Yaskawa INFORM job: A_ROOF_SIDE_0617_2_PAINT_39.JBI

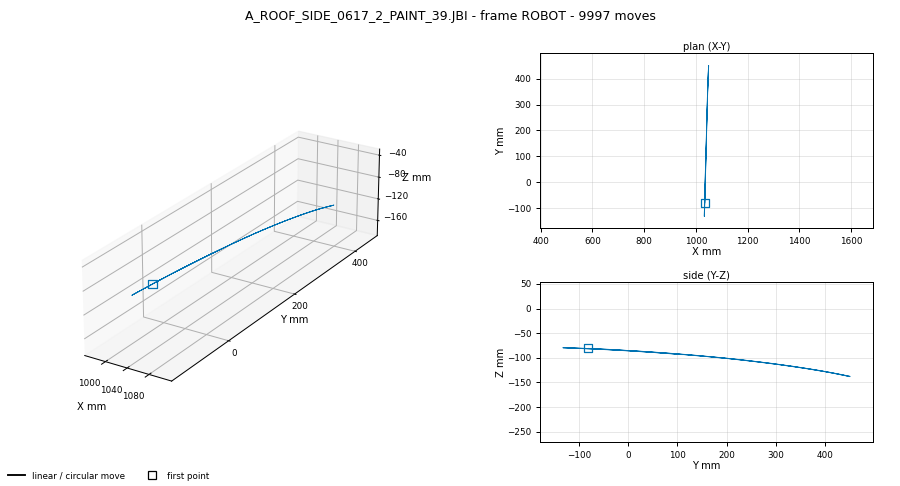
[picture p0: tool path of A_ROOF_SIDE_0617_2_PAINT_39.JBI in frame ROBOT, 9997 of 9997 moves have a stored position in this frame; points joined in program order, loops and branches not executed]
/JOB
//NAME A_ROOF_SIDE_0617_2_PAINT39
//POS
///NPOS 9997,0,0,0,0,0
///TOOL 1
///USER 0
///POSTYPE ROBOT
///RECTAN
///RCONF 1,0,0,0,0,0,0,0,0,0,0,0,0,0,0,0,0,0,0,0,0,0,0,0
C00000=1034.807,-80.393,-80.671,168.125,39.376,157.359
C00001=1034.814,-80.144,-80.681,168.128,39.375,157.359
C00002=1034.820,-79.894,-80.692,168.131,39.374,157.359
C00003=1034.826,-79.644,-80.703,168.134,39.373,157.359
C00004=1034.832,-79.394,-80.715,168.136,39.372,157.359
C00005=1034.838,-79.144,-80.725,168.139,39.372,157.359
C00006=1034.844,-78.895,-80.736,168.142,39.371,157.359
C00007=1034.851,-78.645,-80.747,168.144,39.371,157.359
C00008=1034.856,-78.396,-80.758,168.147,39.370,157.358
C00009=1034.863,-78.145,-80.769,168.150,39.369,157.358
C00010=1034.868,-77.896,-80.780,168.152,39.368,157.358
C00011=1034.875,-77.646,-80.791,168.155,39.368,157.358
C00012=1034.881,-77.397,-80.803,168.157,39.367,157.358
C00013=1034.886,-77.147,-80.814,168.160,39.366,157.358
C00014=1034.893,-76.897,-80.825,168.162,39.365,157.358
C00015=1034.899,-76.648,-80.836,168.165,39.364,157.358
C00016=1034.906,-76.398,-80.846,168.168,39.364,157.358
C00017=1034.911,-76.148,-80.857,168.170,39.363,157.358
C00018=1034.918,-75.899,-80.869,168.173,39.362,157.358
C00019=1034.924,-75.649,-80.880,168.176,39.361,157.358
C00020=1034.930,-75.399,-80.891,168.179,39.361,157.358
C00021=1034.936,-75.150,-80.902,168.181,39.360,157.358
C00022=1034.942,-74.899,-80.914,168.184,39.360,157.358
C00023=1034.948,-74.650,-80.925,168.187,39.359,157.358
C00024=1034.955,-74.400,-80.936,168.189,39.358,157.358
C00025=1034.960,-74.151,-80.947,168.192,39.358,157.358
C00026=1034.967,-73.901,-80.959,168.195,39.357,157.358
C00027=1034.973,-73.652,-80.970,168.196,39.356,157.358
C00028=1034.979,-73.402,-80.981,168.199,39.356,157.358
C00029=1034.985,-73.153,-80.993,168.202,39.355,157.358
C00030=1034.991,-72.902,-81.005,168.204,39.355,157.358
C00031=1034.996,-72.653,-81.016,168.207,39.354,157.358
C00032=1035.002,-72.404,-81.027,168.210,39.354,157.358
C00033=1035.009,-72.154,-81.038,168.212,39.353,157.358
C00034=1035.015,-71.904,-81.049,168.215,39.352,157.358
C00035=1035.020,-71.654,-81.062,168.217,39.352,157.358
C00036=1035.027,-71.404,-81.073,168.220,39.351,157.358
C00037=1035.033,-71.155,-81.085,168.223,39.351,157.358
C00038=1035.039,-70.905,-81.096,168.225,39.350,157.358
C00039=1035.045,-70.656,-81.107,168.228,39.350,157.358
C00040=1035.051,-70.406,-81.119,168.231,39.349,157.358
C00041=1035.057,-70.156,-81.130,168.233,39.348,157.357
C00042=1035.063,-69.907,-81.142,168.236,39.348,157.357
C00043=1035.069,-69.657,-81.153,168.239,39.347,157.357
C00044=1035.076,-69.408,-81.165,168.241,39.347,157.357
C00045=1035.081,-69.158,-81.177,168.244,39.346,157.357
C00046=1035.087,-68.908,-81.188,168.246,39.346,157.357
C00047=1035.094,-68.658,-81.200,168.249,39.345,157.357
C00048=1035.100,-68.375,-81.213,168.251,39.344,157.357
C00049=1035.107,-68.093,-81.226,168.254,39.344,157.357
C00050=1035.114,-67.811,-81.239,168.257,39.343,157.357
C00051=1035.121,-67.528,-81.252,168.260,39.342,157.357
C00052=1035.127,-67.278,-81.264,168.263,39.342,157.357
C00053=1035.133,-67.028,-81.276,168.265,39.341,157.357
C00054=1035.139,-66.778,-81.287,168.268,39.341,157.357
C00055=1035.145,-66.529,-81.299,168.271,39.340,157.357
C00056=1035.152,-66.279,-81.310,168.273,39.340,157.357
C00057=1035.157,-66.029,-81.323,168.276,39.339,157.357
C00058=1035.164,-65.780,-81.334,168.278,39.339,157.357
C00059=1035.170,-65.530,-81.345,168.281,39.338,157.357
C00060=1035.176,-65.281,-81.357,168.284,39.337,157.357
C00061=1035.182,-65.030,-81.369,168.286,39.337,157.357
C00062=1035.188,-64.781,-81.381,168.289,39.336,157.357
C00063=1035.194,-64.532,-81.393,168.292,39.336,157.357
C00064=1035.201,-64.282,-81.404,168.294,39.335,157.357
C00065=1035.206,-64.032,-81.416,168.297,39.335,157.357
C00066=1035.213,-63.783,-81.428,168.299,39.334,157.357
C00067=1035.219,-63.533,-81.439,168.302,39.334,157.357
C00068=1035.226,-63.283,-81.451,168.305,39.333,157.357
C00069=1035.231,-63.034,-81.463,168.307,39.333,157.357
C00070=1035.237,-62.784,-81.475,168.310,39.332,157.357
C00071=1035.244,-62.534,-81.487,168.311,39.331,157.357
C00072=1035.250,-62.285,-81.498,168.314,39.331,157.357
C00073=1035.256,-62.035,-81.511,168.317,39.330,157.357
C00074=1035.262,-61.785,-81.522,168.319,39.330,157.357
C00075=1035.269,-61.536,-81.534,168.322,39.329,157.357
C00076=1035.274,-61.286,-81.546,168.324,39.329,157.357
C00077=1035.281,-61.037,-81.558,168.327,39.328,157.357
C00078=1035.287,-60.787,-81.569,168.330,39.327,157.357
C00079=1035.294,-60.537,-81.581,168.332,39.327,157.357
C00080=1035.299,-60.288,-81.594,168.335,39.326,157.357
C00081=1035.306,-60.038,-81.606,168.338,39.326,157.357
C00082=1035.312,-59.788,-81.617,168.340,39.325,157.357
C00083=1035.318,-59.538,-81.629,168.343,39.325,157.357
C00084=1035.325,-59.289,-81.641,168.345,39.324,157.357
C00085=1035.331,-59.040,-81.653,168.348,39.324,157.357
C00086=1035.337,-58.790,-81.665,168.351,39.323,157.357
C00087=1035.343,-58.540,-81.677,168.353,39.322,157.357
C00088=1035.350,-58.290,-81.689,168.356,39.322,157.357
C00089=1035.356,-58.041,-81.701,168.358,39.321,157.357
C00090=1035.362,-57.791,-81.713,168.361,39.321,157.357
C00091=1035.368,-57.542,-81.725,168.364,39.320,157.357
C00092=1035.375,-57.292,-81.737,168.366,39.320,157.357
C00093=1035.381,-57.042,-81.749,168.369,39.319,157.357
C00094=1035.388,-56.793,-81.761,168.371,39.319,157.357
C00095=1035.394,-56.543,-81.773,168.374,39.318,157.357
C00096=1035.401,-56.294,-81.785,168.375,39.318,157.357
C00097=1035.406,-56.044,-81.797,168.378,39.317,157.357
C00098=1035.412,-55.794,-81.809,168.381,39.316,157.357
C00099=1035.419,-55.545,-81.821,168.383,39.316,157.357
C00100=1035.425,-55.295,-81.833,168.386,39.315,157.357
C00101=1035.432,-55.045,-81.845,168.388,39.315,157.357
C00102=1035.438,-54.796,-81.857,168.391,39.314,157.357
C00103=1035.444,-54.546,-81.870,168.394,39.313,157.357
C00104=1035.451,-54.296,-81.882,168.396,39.313,157.357
C00105=1035.458,-54.047,-81.893,168.399,39.312,157.357
C00106=1035.463,-53.797,-81.906,168.401,39.312,157.357
C00107=1035.469,-53.548,-81.918,168.404,39.311,157.356
C00108=1035.476,-53.298,-81.930,168.407,39.311,157.357
C00109=1035.482,-53.048,-81.942,168.409,39.310,157.356
C00110=1035.489,-52.799,-81.954,168.412,39.310,157.357
C00111=1035.495,-52.549,-81.966,168.414,39.309,157.356
C00112=1035.503,-52.268,-81.980,168.417,39.309,157.356
C00113=1035.510,-51.986,-81.994,168.420,39.308,157.356
C00114=1035.516,-51.705,-82.008,168.423,39.307,157.356
C00115=1035.524,-51.423,-82.021,168.426,39.307,157.356
C00116=1035.530,-51.174,-82.034,168.428,39.306,157.356
C00117=1035.537,-50.924,-82.046,168.431,39.306,157.356
C00118=1035.543,-50.674,-82.058,168.434,39.305,157.356
C00119=1035.549,-50.424,-82.070,168.436,39.305,157.356
C00120=1035.556,-50.175,-82.084,168.439,39.305,157.356
C00121=1035.562,-49.926,-82.096,168.440,39.304,157.356
C00122=1035.568,-49.676,-82.108,168.444,39.304,157.356
C00123=1035.574,-49.426,-82.121,168.446,39.304,157.356
C00124=1035.581,-49.176,-82.133,168.449,39.304,157.357
C00125=1035.587,-48.927,-82.146,168.450,39.303,157.356
C00126=1035.593,-48.677,-82.159,168.453,39.303,157.356
C00127=1035.598,-48.428,-82.171,168.456,39.302,157.357
C00128=1035.605,-48.178,-82.183,168.459,39.302,157.357
C00129=1035.611,-47.929,-82.196,168.460,39.301,157.356
C00130=1035.617,-47.679,-82.208,168.463,39.301,157.357
C00131=1035.624,-47.430,-82.220,168.465,39.301,157.357
C00132=1035.630,-47.180,-82.234,168.468,39.300,157.357
C00133=1035.636,-46.931,-82.246,168.470,39.300,157.357
C00134=1035.642,-46.681,-82.259,168.473,39.300,157.357
C00135=1035.649,-46.432,-82.271,168.475,39.300,157.357
C00136=1035.654,-46.182,-82.284,168.478,39.299,157.357
C00137=1035.660,-45.932,-82.297,168.480,39.299,157.357
C00138=1035.667,-45.683,-82.310,168.483,39.298,157.357
C00139=1035.673,-45.433,-82.322,168.485,39.298,157.357
C00140=1035.679,-45.183,-82.334,168.488,39.297,157.357
C00141=1035.686,-44.933,-82.348,168.490,39.297,157.357
C00142=1035.693,-44.684,-82.360,168.493,39.297,157.357
C00143=1035.698,-44.434,-82.373,168.495,39.297,157.357
C00144=1035.705,-44.185,-82.386,168.498,39.296,157.357
C00145=1035.711,-43.935,-82.398,168.500,39.296,157.357
C00146=1035.718,-43.686,-82.411,168.503,39.296,157.357
C00147=1035.723,-43.436,-82.424,168.505,39.295,157.357
C00148=1035.729,-43.186,-82.436,168.507,39.295,157.357
C00149=1035.736,-42.937,-82.449,168.510,39.294,157.357
C00150=1035.742,-42.687,-82.461,168.512,39.294,157.357
C00151=1035.748,-42.438,-82.475,168.515,39.293,157.357
C00152=1035.754,-42.188,-82.487,168.517,39.293,157.357
C00153=1035.761,-41.939,-82.500,168.520,39.293,157.357
C00154=1035.768,-41.688,-82.513,168.522,39.293,157.357
C00155=1035.774,-41.439,-82.526,168.525,39.292,157.357
C00156=1035.780,-41.189,-82.539,168.527,39.292,157.357
C00157=1035.786,-40.940,-82.552,168.530,39.292,157.357
C00158=1035.793,-40.690,-82.564,168.532,39.292,157.357
C00159=1035.799,-40.441,-82.577,168.535,39.291,157.357
C00160=1035.805,-40.191,-82.590,168.537,39.291,157.357
C00161=1035.812,-39.941,-82.603,168.540,39.290,157.357
C00162=1035.818,-39.691,-82.616,168.542,39.290,157.357
C00163=1035.825,-39.442,-82.629,168.545,39.289,157.357
C00164=1035.831,-39.193,-82.641,168.547,39.289,157.357
C00165=1035.837,-38.943,-82.654,168.550,39.289,157.357
C00166=1035.843,-38.694,-82.668,168.552,39.289,157.357
C00167=1035.849,-38.443,-82.681,168.554,39.288,157.357
C00168=1035.856,-38.194,-82.694,168.557,39.288,157.357
C00169=1035.862,-37.944,-82.706,168.559,39.288,157.357
C00170=1035.868,-37.695,-82.720,168.562,39.287,157.357
C00171=1035.874,-37.446,-82.733,168.564,39.287,157.357
C00172=1035.880,-37.196,-82.745,168.567,39.287,157.357
C00173=1035.886,-36.947,-82.759,168.569,39.287,157.357
C00174=1035.893,-36.697,-82.772,168.571,39.287,157.357
C00175=1035.899,-36.447,-82.786,168.574,39.287,157.357
C00176=1035.906,-36.167,-82.800,168.576,39.286,157.357
C00177=1035.913,-35.885,-82.815,168.579,39.286,157.357
C00178=1035.920,-35.604,-82.830,168.582,39.285,157.357
C00179=1035.928,-35.323,-82.844,168.585,39.285,157.358
C00180=1035.934,-35.074,-82.858,168.587,39.285,157.358
C00181=1035.940,-34.824,-82.871,168.589,39.285,157.358
C00182=1035.946,-34.574,-82.883,168.592,39.285,157.358
C00183=1035.952,-34.325,-82.897,168.594,39.284,157.358
C00184=1035.959,-34.075,-82.910,168.597,39.284,157.358
C00185=1035.964,-33.826,-82.924,168.599,39.284,157.358
C00186=1035.971,-33.576,-82.937,168.601,39.283,157.358
C00187=1035.977,-33.326,-82.950,168.604,39.283,157.358
C00188=1035.983,-33.076,-82.964,168.606,39.283,157.358
C00189=1035.990,-32.827,-82.977,168.609,39.283,157.358
C00190=1035.996,-32.578,-82.990,168.611,39.283,157.358
C00191=1036.002,-32.329,-83.003,168.614,39.282,157.358
C00192=1036.008,-32.078,-83.016,168.616,39.282,157.358
C00193=1036.015,-31.829,-83.030,168.618,39.282,157.358
C00194=1036.021,-31.580,-83.043,168.621,39.282,157.358
C00195=1036.028,-31.330,-83.057,168.623,39.281,157.358
C00196=1036.034,-31.080,-83.070,168.626,39.281,157.358
C00197=1036.040,-30.831,-83.083,168.628,39.281,157.358
C00198=1036.046,-30.582,-83.096,168.630,39.281,157.358
C00199=1036.053,-30.332,-83.110,168.633,39.280,157.358
C00200=1036.059,-30.082,-83.123,168.635,39.280,157.358
C00201=1036.065,-29.833,-83.136,168.637,39.280,157.358
C00202=1036.072,-29.583,-83.149,168.640,39.280,157.358
C00203=1036.078,-29.333,-83.163,168.643,39.280,157.358
C00204=1036.084,-29.084,-83.177,168.645,39.279,157.358
C00205=1036.091,-28.834,-83.190,168.647,39.279,157.358
C00206=1036.097,-28.585,-83.203,168.649,39.279,157.358
C00207=1036.103,-28.335,-83.217,168.652,39.278,157.358
C00208=1036.110,-28.085,-83.230,168.654,39.278,157.358
C00209=1036.116,-27.836,-83.244,168.658,39.278,157.359
C00210=1036.123,-27.586,-83.257,168.660,39.278,157.359
C00211=1036.129,-27.337,-83.271,168.662,39.278,157.359
C00212=1036.135,-27.088,-83.284,168.665,39.277,157.359
C00213=1036.142,-26.838,-83.297,168.667,39.277,157.359
C00214=1036.148,-26.588,-83.311,168.669,39.277,157.359
C00215=1036.154,-26.339,-83.325,168.672,39.277,157.359
C00216=1036.161,-26.089,-83.338,168.674,39.277,157.359
C00217=1036.166,-25.839,-83.352,168.676,39.277,157.359
C00218=1036.172,-25.590,-83.365,168.679,39.276,157.359
C00219=1036.179,-25.341,-83.380,168.681,39.276,157.359
C00220=1036.185,-25.091,-83.394,168.683,39.276,157.359
C00221=1036.192,-24.841,-83.407,168.686,39.276,157.359
C00222=1036.198,-24.592,-83.420,168.688,39.276,157.359
C00223=1036.203,-24.342,-83.434,168.690,39.276,157.359
C00224=1036.210,-24.092,-83.448,168.693,39.275,157.359
C00225=1036.216,-23.843,-83.461,168.695,39.275,157.359
C00226=1036.223,-23.593,-83.476,168.697,39.275,157.359
C00227=1036.229,-23.344,-83.489,168.700,39.275,157.359
C00228=1036.235,-23.095,-83.503,168.702,39.275,157.359
C00229=1036.241,-22.845,-83.517,168.704,39.275,157.359
C00230=1036.248,-22.595,-83.530,168.707,39.274,157.359
C00231=1036.255,-22.346,-83.545,168.709,39.274,157.359
C00232=1036.264,-21.949,-83.566,168.713,39.275,157.360
C00233=1036.274,-21.552,-83.588,168.716,39.274,157.360
C00234=1036.284,-21.155,-83.611,168.720,39.274,157.360
C00235=1036.294,-20.758,-83.632,168.724,39.274,157.360
C00236=1036.304,-20.374,-83.654,168.727,39.274,157.360
C00237=1036.314,-19.990,-83.675,168.731,39.273,157.360
C00238=1036.323,-19.606,-83.696,168.735,39.273,157.360
C00239=1036.333,-19.222,-83.718,168.738,39.273,157.360
C00240=1036.339,-18.973,-83.732,168.740,39.273,157.360
C00241=1036.346,-18.723,-83.745,168.743,39.272,157.360
C00242=1036.352,-18.474,-83.759,168.745,39.272,157.360
C00243=1036.358,-18.224,-83.773,168.747,39.272,157.360
C00244=1036.365,-17.975,-83.787,168.750,39.272,157.360
C00245=1036.371,-17.725,-83.802,168.753,39.272,157.360
C00246=1036.377,-17.476,-83.815,168.755,39.272,157.360
C00247=1036.384,-17.226,-83.829,168.758,39.271,157.360
C00248=1036.390,-16.977,-83.843,168.760,39.271,157.361
C00249=1036.397,-16.727,-83.857,168.762,39.271,157.361
C00250=1036.403,-16.477,-83.872,168.765,39.271,157.361
C00251=1036.409,-16.228,-83.885,168.767,39.271,157.361
C00252=1036.416,-15.979,-83.899,168.769,39.271,157.361
C00253=1036.422,-15.729,-83.913,168.771,39.271,157.361
C00254=1036.429,-15.479,-83.927,168.774,39.270,157.361
C00255=1036.434,-15.230,-83.941,168.776,39.270,157.361
C00256=1036.441,-14.980,-83.955,168.778,39.271,157.361
C00257=1036.447,-14.731,-83.970,168.781,39.270,157.361
C00258=1036.454,-14.481,-83.983,168.783,39.270,157.361
C00259=1036.460,-14.231,-83.998,168.785,39.270,157.361
C00260=1036.466,-13.982,-84.012,168.787,39.270,157.361
C00261=1036.473,-13.733,-84.026,168.790,39.270,157.361
C00262=1036.478,-13.483,-84.040,168.792,39.270,157.361
C00263=1036.485,-13.233,-84.055,168.794,39.270,157.361
C00264=1036.491,-12.985,-84.069,168.796,39.270,157.361
C00265=1036.497,-12.734,-84.083,168.799,39.270,157.361
C00266=1036.504,-12.485,-84.098,168.801,39.270,157.362
C00267=1036.510,-12.235,-84.112,168.803,39.270,157.362
C00268=1036.516,-11.986,-84.127,168.805,39.270,157.362
C00269=1036.522,-11.737,-84.140,168.808,39.270,157.362
C00270=1036.529,-11.487,-84.155,168.810,39.270,157.362
C00271=1036.535,-11.237,-84.170,168.812,39.270,157.362
C00272=1036.541,-10.988,-84.183,168.814,39.269,157.362
C00273=1036.548,-10.738,-84.198,168.818,39.270,157.362
C00274=1036.554,-10.489,-84.213,168.820,39.270,157.362
C00275=1036.560,-10.239,-84.226,168.822,39.270,157.362
C00276=1036.567,-9.990,-84.241,168.824,39.269,157.362
C00277=1036.573,-9.741,-84.256,168.827,39.269,157.362
C00278=1036.579,-9.491,-84.269,168.829,39.269,157.362
C00279=1036.586,-9.241,-84.284,168.831,39.270,157.362
C00280=1036.592,-8.992,-84.299,168.833,39.269,157.362
C00281=1036.598,-8.742,-84.312,168.836,39.269,157.362
C00282=1036.605,-8.493,-84.327,168.838,39.269,157.363
C00283=1036.611,-8.244,-84.342,168.840,39.269,157.363
C00284=1036.617,-7.994,-84.356,168.842,39.269,157.363
C00285=1036.624,-7.744,-84.371,168.844,39.269,157.363
C00286=1036.630,-7.495,-84.385,168.847,39.269,157.363
C00287=1036.637,-7.246,-84.400,168.849,39.269,157.363
C00288=1036.643,-6.995,-84.414,168.851,39.269,157.363
C00289=1036.648,-6.746,-84.428,168.853,39.269,157.363
C00290=1036.656,-6.497,-84.443,168.856,39.268,157.363
C00291=1036.662,-6.247,-84.458,168.858,39.268,157.363
C00292=1036.668,-5.997,-84.472,168.860,39.269,157.363
C00293=1036.675,-5.749,-84.486,168.862,39.269,157.363
C00294=1036.681,-5.499,-84.501,168.865,39.268,157.363
C00295=1036.687,-5.249,-84.516,168.867,39.268,157.363
C00296=1036.694,-5.001,-84.530,168.869,39.268,157.363
C00297=1036.700,-4.750,-84.544,168.871,39.268,157.363
C00298=1036.706,-4.501,-84.559,168.873,39.268,157.363
C00299=1036.713,-4.251,-84.573,168.877,39.268,157.364
C00300=1036.721,-3.968,-84.590,168.879,39.268,157.364
C00301=1036.728,-3.685,-84.607,168.882,39.268,157.364
C00302=1036.734,-3.401,-84.624,168.884,39.268,157.364
C00303=1036.741,-3.118,-84.640,168.887,39.268,157.364
C00304=1036.748,-2.868,-84.655,168.889,39.268,157.364
C00305=1036.754,-2.618,-84.670,168.891,39.268,157.364
C00306=1036.760,-2.369,-84.685,168.893,39.268,157.364
C00307=1036.766,-2.120,-84.699,168.895,39.268,157.364
C00308=1036.773,-1.870,-84.714,168.898,39.268,157.364
C00309=1036.779,-1.620,-84.729,168.900,39.269,157.364
C00310=1036.785,-1.372,-84.744,168.902,39.268,157.364
C00311=1036.791,-1.122,-84.759,168.904,39.268,157.364
C00312=1036.798,-0.872,-84.774,168.906,39.269,157.365
C00313=1036.804,-0.623,-84.789,168.908,39.269,157.365
C00314=1036.810,-0.373,-84.804,168.911,39.268,157.365
C00315=1036.816,-0.124,-84.818,168.914,39.269,157.365
C00316=1036.823,0.126,-84.833,168.916,39.269,157.365
C00317=1036.829,0.375,-84.848,168.918,39.269,157.365
C00318=1036.835,0.625,-84.863,168.920,39.269,157.365
C00319=1036.841,0.874,-84.878,168.922,39.269,157.365
C00320=1036.847,1.124,-84.893,168.924,39.269,157.365
C00321=1036.854,1.373,-84.908,168.927,39.269,157.365
C00322=1036.860,1.623,-84.922,168.929,39.269,157.365
C00323=1036.867,1.872,-84.938,168.931,39.269,157.365
C00324=1036.873,2.121,-84.953,168.933,39.270,157.366
C00325=1036.879,2.371,-84.968,168.935,39.269,157.366
C00326=1036.885,2.620,-84.983,168.937,39.269,157.366
C00327=1036.892,2.870,-84.998,168.940,39.270,157.366
C00328=1036.898,3.120,-85.013,168.942,39.270,157.366
C00329=1036.904,3.370,-85.028,168.944,39.269,157.366
C00330=1036.910,3.619,-85.043,168.946,39.270,157.366
C00331=1036.916,3.868,-85.058,168.948,39.270,157.366
C00332=1036.923,4.117,-85.073,168.950,39.270,157.366
C00333=1036.929,4.367,-85.088,168.953,39.270,157.366
C00334=1036.935,4.617,-85.103,168.956,39.270,157.366
C00335=1036.942,4.866,-85.118,168.958,39.270,157.366
C00336=1036.948,5.116,-85.133,168.960,39.270,157.366
C00337=1036.954,5.364,-85.148,168.962,39.270,157.367
C00338=1036.961,5.614,-85.163,168.964,39.270,157.367
C00339=1036.967,5.863,-85.178,168.966,39.270,157.367
C00340=1036.973,6.113,-85.193,168.969,39.270,157.367
C00341=1036.980,6.362,-85.209,168.971,39.270,157.367
C00342=1036.987,6.612,-85.224,168.973,39.270,157.367
C00343=1036.993,6.861,-85.239,168.975,39.270,157.367
C00344=1036.999,7.111,-85.254,168.977,39.270,157.367
C00345=1037.006,7.360,-85.269,168.979,39.270,157.367
C00346=1037.012,7.610,-85.284,168.981,39.270,157.367
C00347=1037.018,7.860,-85.300,168.984,39.270,157.367
C00348=1037.024,8.109,-85.314,168.986,39.270,157.367
C00349=1037.031,8.358,-85.330,168.988,39.270,157.367
C00350=1037.037,8.607,-85.345,168.991,39.271,157.368
C00351=1037.043,8.857,-85.360,168.993,39.271,157.368
C00352=1037.050,9.106,-85.376,168.995,39.270,157.368
C00353=1037.056,9.356,-85.391,168.997,39.270,157.368
C00354=1037.063,9.605,-85.405,169.000,39.271,157.368
C00355=1037.069,9.854,-85.421,169.002,39.271,157.368
C00356=1037.076,10.104,-85.436,169.004,39.270,157.368
C00357=1037.082,10.354,-85.451,169.006,39.271,157.368
C00358=1037.089,10.603,-85.467,169.008,39.271,157.368
C00359=1037.095,10.853,-85.482,169.010,39.271,157.368
C00360=1037.101,11.102,-85.497,169.012,39.270,157.368
C00361=1037.108,11.352,-85.513,169.014,39.271,157.368
C00362=1037.114,11.601,-85.528,169.017,39.271,157.368
C00363=1037.120,11.851,-85.543,169.019,39.271,157.368
C00364=1037.128,12.136,-85.560,169.021,39.271,157.369
C00365=1037.135,12.421,-85.578,169.024,39.271,157.369
C00366=1037.143,12.706,-85.596,169.026,39.271,157.369
C00367=1037.150,12.992,-85.613,169.029,39.271,157.369
C00368=1037.157,13.241,-85.628,169.032,39.271,157.369
C00369=1037.163,13.491,-85.643,169.034,39.271,157.369
C00370=1037.170,13.740,-85.659,169.036,39.271,157.369
C00371=1037.176,13.990,-85.675,169.038,39.271,157.369
C00372=1037.182,14.239,-85.690,169.040,39.271,157.369
C00373=1037.189,14.489,-85.705,169.042,39.271,157.369
C00374=1037.195,14.738,-85.721,169.044,39.271,157.369
C00375=1037.201,14.988,-85.736,169.046,39.271,157.369
C00376=1037.208,15.237,-85.752,169.048,39.272,157.370
C00377=1037.214,15.486,-85.768,169.051,39.272,157.370
C00378=1037.220,15.736,-85.783,169.053,39.271,157.370
C00379=1037.227,15.985,-85.799,169.055,39.272,157.370
C00380=1037.232,16.235,-85.814,169.057,39.272,157.370
C00381=1037.239,16.484,-85.830,169.059,39.272,157.370
C00382=1037.245,16.734,-85.846,169.061,39.272,157.370
C00383=1037.251,16.983,-85.861,169.063,39.272,157.370
C00384=1037.258,17.232,-85.877,169.066,39.273,157.370
C00385=1037.264,17.482,-85.893,169.068,39.272,157.370
C00386=1037.271,17.732,-85.909,169.070,39.273,157.370
C00387=1037.278,17.981,-85.924,169.072,39.273,157.371
C00388=1037.283,18.231,-85.940,169.074,39.273,157.371
C00389=1037.290,18.480,-85.955,169.077,39.273,157.371
C00390=1037.297,18.729,-85.971,169.079,39.273,157.371
C00391=1037.302,18.979,-85.987,169.081,39.273,157.371
C00392=1037.309,19.228,-86.002,169.083,39.273,157.371
C00393=1037.315,19.477,-86.019,169.085,39.273,157.371
C00394=1037.321,19.727,-86.033,169.087,39.274,157.371
C00395=1037.328,19.976,-86.049,169.089,39.273,157.371
C00396=1037.335,20.226,-86.066,169.091,39.274,157.371
C00397=1037.341,20.475,-86.081,169.093,39.274,157.371
C00398=1037.347,20.725,-86.097,169.095,39.274,157.371
C00399=1037.354,20.974,-86.113,169.098,39.274,157.372
C00400=1037.360,21.223,-86.129,169.100,39.274,157.372
C00401=1037.366,21.473,-86.144,169.102,39.275,157.372
C00402=1037.372,21.722,-86.160,169.104,39.274,157.372
C00403=1037.378,21.971,-86.176,169.106,39.275,157.372
C00404=1037.385,22.221,-86.192,169.109,39.275,157.372
C00405=1037.391,22.471,-86.209,169.111,39.275,157.372
C00406=1037.398,22.720,-86.224,169.113,39.275,157.372
C00407=1037.403,22.970,-86.240,169.115,39.276,157.372
C00408=1037.410,23.219,-86.255,169.117,39.275,157.372
C00409=1037.416,23.468,-86.272,169.119,39.275,157.372
C00410=1037.423,23.717,-86.287,169.121,39.276,157.373
C00411=1037.429,23.966,-86.304,169.123,39.276,157.373
C00412=1037.436,24.217,-86.319,169.126,39.276,157.373
C00413=1037.442,24.466,-86.335,169.128,39.276,157.373
C00414=1037.448,24.715,-86.351,169.130,39.277,157.373
C00415=1037.454,24.964,-86.367,169.132,39.276,157.373
C00416=1037.461,25.213,-86.383,169.134,39.276,157.373
C00417=1037.467,25.463,-86.399,169.136,39.277,157.373
C00418=1037.474,25.713,-86.415,169.138,39.277,157.373
C00419=1037.480,25.962,-86.431,169.140,39.277,157.373
C00420=1037.486,26.211,-86.448,169.142,39.277,157.373
C00421=1037.493,26.461,-86.463,169.144,39.277,157.374
C00422=1037.499,26.711,-86.479,169.146,39.277,157.374
C00423=1037.506,26.960,-86.495,169.149,39.278,157.374
C00424=1037.512,27.209,-86.511,169.151,39.278,157.374
C00425=1037.518,27.459,-86.527,169.153,39.277,157.374
C00426=1037.524,27.708,-86.543,169.156,39.278,157.374
C00427=1037.531,27.958,-86.560,169.158,39.278,157.374
C00428=1037.538,28.244,-86.578,169.160,39.278,157.374
C00429=1037.545,28.531,-86.596,169.162,39.278,157.374
C00430=1037.553,28.817,-86.615,169.165,39.279,157.374
C00431=1037.559,29.104,-86.634,169.167,39.279,157.375
C00432=1037.567,29.353,-86.650,169.169,39.279,157.375
C00433=1037.573,29.603,-86.666,169.171,39.279,157.375
C00434=1037.579,29.852,-86.683,169.173,39.279,157.375
C00435=1037.585,30.101,-86.699,169.175,39.280,157.375
C00436=1037.592,30.351,-86.715,169.177,39.280,157.375
C00437=1037.598,30.601,-86.731,169.179,39.280,157.375
C00438=1037.604,30.850,-86.747,169.182,39.280,157.375
C00439=1037.610,31.099,-86.764,169.184,39.280,157.375
C00440=1037.616,31.348,-86.781,169.186,39.280,157.375
C00441=1037.623,31.598,-86.797,169.188,39.281,157.376
C00442=1037.629,31.847,-86.813,169.190,39.281,157.376
C00443=1037.635,32.096,-86.829,169.192,39.281,157.376
C00444=1037.642,32.346,-86.846,169.194,39.281,157.376
C00445=1037.648,32.596,-86.861,169.196,39.282,157.376
C00446=1037.654,32.845,-86.878,169.198,39.281,157.376
C00447=1037.661,33.094,-86.895,169.200,39.282,157.376
C00448=1037.667,33.344,-86.911,169.202,39.282,157.376
C00449=1037.673,33.593,-86.928,169.204,39.282,157.376
C00450=1037.680,33.842,-86.943,169.207,39.283,157.377
C00451=1037.686,34.092,-86.960,169.209,39.283,157.377
C00452=1037.693,34.341,-86.977,169.211,39.283,157.377
C00453=1037.699,34.590,-86.993,169.213,39.283,157.377
C00454=1037.706,34.840,-87.009,169.215,39.283,157.377
C00455=1037.712,35.089,-87.025,169.217,39.283,157.377
C00456=1037.718,35.339,-87.042,169.219,39.283,157.377
C00457=1037.725,35.588,-87.059,169.221,39.284,157.377
C00458=1037.731,35.837,-87.075,169.223,39.284,157.377
C00459=1037.737,36.086,-87.091,169.225,39.284,157.377
C00460=1037.744,36.336,-87.108,169.227,39.284,157.377
C00461=1037.750,36.585,-87.124,169.229,39.284,157.378
C00462=1037.756,36.835,-87.141,169.231,39.284,157.378
C00463=1037.763,37.085,-87.157,169.234,39.285,157.378
C00464=1037.769,37.333,-87.174,169.236,39.285,157.378
C00465=1037.775,37.583,-87.191,169.238,39.285,157.378
C00466=1037.781,37.833,-87.207,169.240,39.286,157.378
C00467=1037.788,38.081,-87.224,169.242,39.285,157.378
C00468=1037.794,38.332,-87.241,169.244,39.286,157.378
C00469=1037.800,38.581,-87.257,169.246,39.286,157.378
C00470=1037.806,38.830,-87.274,169.248,39.286,157.379
C00471=1037.813,39.080,-87.291,169.250,39.287,157.379
C00472=1037.819,39.329,-87.307,169.252,39.287,157.379
C00473=1037.825,39.578,-87.324,169.254,39.287,157.379
C00474=1037.832,39.828,-87.341,169.257,39.287,157.379
C00475=1037.838,40.076,-87.357,169.259,39.288,157.379
C00476=1037.844,40.326,-87.374,169.261,39.287,157.379
C00477=1037.851,40.575,-87.391,169.263,39.288,157.379
C00478=1037.857,40.825,-87.407,169.265,39.288,157.379
C00479=1037.863,41.075,-87.424,169.267,39.288,157.379
C00480=1037.870,41.323,-87.441,169.269,39.289,157.380
C00481=1037.875,41.573,-87.457,169.271,39.289,157.380
C00482=1037.882,41.822,-87.475,169.273,39.289,157.380
C00483=1037.888,42.072,-87.491,169.275,39.290,157.380
C00484=1037.895,42.321,-87.508,169.277,39.289,157.380
C00485=1037.901,42.570,-87.524,169.280,39.290,157.380
C00486=1037.907,42.819,-87.541,169.282,39.290,157.380
C00487=1037.914,43.069,-87.558,169.284,39.290,157.380
C00488=1037.920,43.318,-87.575,169.286,39.290,157.380
C00489=1037.926,43.568,-87.592,169.288,39.291,157.381
C00490=1037.932,43.817,-87.609,169.290,39.291,157.381
C00491=1037.939,44.067,-87.626,169.292,39.292,157.381
C00492=1037.946,44.353,-87.646,169.294,39.291,157.381
C00493=1037.952,44.639,-87.665,169.296,39.292,157.381
C00494=1037.960,44.926,-87.685,169.298,39.292,157.381
C00495=1037.967,45.213,-87.704,169.302,39.293,157.381
C00496=1037.973,45.461,-87.721,169.304,39.293,157.382
C00497=1037.979,45.711,-87.738,169.305,39.293,157.382
C00498=1037.985,45.960,-87.756,169.307,39.294,157.382
C00499=1037.992,46.210,-87.773,169.309,39.294,157.382
C00500=1037.998,46.459,-87.789,169.311,39.294,157.382
C00501=1038.005,46.709,-87.807,169.313,39.295,157.382
C00502=1038.010,46.958,-87.824,169.315,39.295,157.382
C00503=1038.016,47.207,-87.840,169.317,39.295,157.382
C00504=1038.023,47.456,-87.858,169.320,39.296,157.382
C00505=1038.028,47.706,-87.875,169.322,39.296,157.383
C00506=1038.035,47.956,-87.892,169.324,39.296,157.383
C00507=1038.041,48.204,-87.909,169.326,39.296,157.383
C00508=1038.047,48.454,-87.927,169.328,39.297,157.383
C00509=1038.054,48.703,-87.944,169.330,39.297,157.383
C00510=1038.060,48.953,-87.960,169.332,39.297,157.383
C00511=1038.066,49.202,-87.978,169.334,39.298,157.383
C00512=1038.073,49.451,-87.995,169.336,39.298,157.384
C00513=1038.079,49.701,-88.012,169.337,39.298,157.384
C00514=1038.085,49.950,-88.030,169.340,39.299,157.384
C00515=1038.091,50.199,-88.047,169.342,39.299,157.384
C00516=1038.098,50.449,-88.064,169.344,39.299,157.384
C00517=1038.104,50.697,-88.081,169.346,39.300,157.384
C00518=1038.110,50.948,-88.098,169.348,39.300,157.384
C00519=1038.116,51.196,-88.115,169.350,39.300,157.384
C00520=1038.123,51.446,-88.132,169.352,39.300,157.384
C00521=1038.128,51.695,-88.150,169.354,39.300,157.384
C00522=1038.135,51.944,-88.167,169.356,39.301,157.385
C00523=1038.142,52.194,-88.184,169.358,39.301,157.385
C00524=1038.147,52.443,-88.201,169.360,39.301,157.385
C00525=1038.154,52.693,-88.219,169.363,39.302,157.385
C00526=1038.161,52.942,-88.236,169.365,39.302,157.385
C00527=1038.167,53.191,-88.254,169.367,39.302,157.385
C00528=1038.173,53.440,-88.271,169.369,39.302,157.385
C00529=1038.179,53.690,-88.289,169.371,39.303,157.385
C00530=1038.185,53.939,-88.305,169.373,39.303,157.386
C00531=1038.192,54.189,-88.322,169.375,39.303,157.386
C00532=1038.198,54.438,-88.340,169.376,39.304,157.386
C00533=1038.204,54.687,-88.357,169.378,39.304,157.386
C00534=1038.211,54.936,-88.374,169.381,39.304,157.386
C00535=1038.217,55.185,-88.392,169.383,39.304,157.386
C00536=1038.223,55.435,-88.409,169.385,39.305,157.386
C00537=1038.230,55.684,-88.427,169.387,39.305,157.386
C00538=1038.236,55.933,-88.444,169.389,39.305,157.386
C00539=1038.243,56.183,-88.462,169.391,39.305,157.387
C00540=1038.250,56.432,-88.479,169.393,39.305,157.387
C00541=1038.255,56.681,-88.496,169.395,39.306,157.387
C00542=1038.262,56.931,-88.514,169.397,39.306,157.387
C00543=1038.267,57.180,-88.531,169.399,39.306,157.387
C00544=1038.274,57.429,-88.549,169.401,39.307,157.387
C00545=1038.281,57.679,-88.565,169.404,39.307,157.387
C00546=1038.286,57.928,-88.583,169.406,39.307,157.387
C00547=1038.293,58.178,-88.600,169.408,39.307,157.387
C00548=1038.300,58.427,-88.618,169.410,39.307,157.388
C00549=1038.306,58.676,-88.636,169.412,39.308,157.388
C00550=1038.313,58.925,-88.653,169.414,39.308,157.388
C00551=1038.320,59.174,-88.671,169.416,39.308,157.388
C00552=1038.325,59.423,-88.688,169.418,39.309,157.388
C00553=1038.332,59.673,-88.705,169.419,39.309,157.388
C00554=1038.338,59.923,-88.723,169.421,39.309,157.388
C00555=1038.345,60.172,-88.741,169.423,39.309,157.388
C00556=1038.352,60.458,-88.761,169.427,39.309,157.388
C00557=1038.360,60.745,-88.781,169.429,39.310,157.389
C00558=1038.366,61.031,-88.801,169.431,39.310,157.389
C00559=1038.374,61.317,-88.821,169.433,39.310,157.389
C00560=1038.380,61.566,-88.838,169.435,39.311,157.389
C00561=1038.387,61.815,-88.856,169.437,39.310,157.389
C00562=1038.393,62.065,-88.874,169.439,39.311,157.389
C00563=1038.400,62.315,-88.891,169.441,39.311,157.389
C00564=1038.406,62.564,-88.908,169.443,39.311,157.389
C00565=1038.413,62.812,-88.926,169.445,39.311,157.389
C00566=1038.420,63.062,-88.944,169.447,39.312,157.390
C00567=1038.426,63.312,-88.962,169.450,39.312,157.390
C00568=1038.432,63.560,-88.979,169.452,39.312,157.390
C00569=1038.438,63.810,-88.997,169.454,39.312,157.390
C00570=1038.445,64.059,-89.014,169.456,39.312,157.390
C00571=1038.451,64.309,-89.033,169.458,39.313,157.390
C00572=1038.457,64.558,-89.050,169.460,39.313,157.390
C00573=1038.464,64.807,-89.068,169.462,39.314,157.390
C00574=1038.470,65.057,-89.085,169.464,39.314,157.390
C00575=1038.476,65.306,-89.104,169.466,39.314,157.391
C00576=1038.483,65.555,-89.121,169.468,39.315,157.391
C00577=1038.489,65.804,-89.139,169.470,39.315,157.391
C00578=1038.495,66.053,-89.158,169.472,39.315,157.391
C00579=1038.502,66.303,-89.175,169.474,39.316,157.391
C00580=1038.508,66.552,-89.193,169.476,39.315,157.391
C00581=1038.514,66.802,-89.211,169.478,39.316,157.391
C00582=1038.521,67.050,-89.229,169.480,39.316,157.391
C00583=1038.527,67.300,-89.246,169.482,39.317,157.392
C00584=1038.532,67.549,-89.264,169.484,39.317,157.392
C00585=1038.539,67.798,-89.283,169.486,39.317,157.392
C00586=1038.546,68.048,-89.300,169.489,39.318,157.392
C00587=1038.552,68.297,-89.319,169.491,39.318,157.392
C00588=1038.558,68.546,-89.336,169.493,39.318,157.392
C00589=1038.565,68.795,-89.354,169.494,39.319,157.392
C00590=1038.571,69.045,-89.372,169.496,39.319,157.393
C00591=1038.577,69.294,-89.390,169.498,39.319,157.393
C00592=1038.584,69.543,-89.409,169.500,39.320,157.393
C00593=1038.589,69.792,-89.426,169.502,39.320,157.393
C00594=1038.596,70.042,-89.444,169.504,39.320,157.393
C00595=1038.602,70.291,-89.462,169.506,39.320,157.393
C00596=1038.608,70.541,-89.480,169.509,39.321,157.393
C00597=1038.615,70.790,-89.499,169.511,39.321,157.393
C00598=1038.620,71.039,-89.517,169.513,39.322,157.394
C00599=1038.627,71.288,-89.535,169.515,39.322,157.394
C00600=1038.633,71.538,-89.553,169.517,39.322,157.394
C00601=1038.640,71.787,-89.571,169.518,39.323,157.394
C00602=1038.646,72.036,-89.589,169.520,39.323,157.394
C00603=1038.652,72.285,-89.607,169.522,39.323,157.394
C00604=1038.658,72.534,-89.625,169.524,39.324,157.394
C00605=1038.665,72.784,-89.644,169.527,39.324,157.394
C00606=1038.671,73.033,-89.662,169.529,39.325,157.395
C00607=1038.677,73.282,-89.681,169.531,39.324,157.395
C00608=1038.683,73.532,-89.698,169.533,39.325,157.395
C00609=1038.689,73.781,-89.717,169.535,39.325,157.395
C00610=1038.696,74.030,-89.735,169.537,39.326,157.395
C00611=1038.702,74.279,-89.753,169.539,39.326,157.395
C00612=1038.709,74.528,-89.771,169.540,39.326,157.395
C00613=1038.715,74.778,-89.789,169.543,39.327,157.395
C00614=1038.721,75.027,-89.808,169.545,39.327,157.396
C00615=1038.728,75.276,-89.827,169.547,39.327,157.396
C00616=1038.733,75.525,-89.844,169.549,39.328,157.396
C00617=1038.740,75.774,-89.863,169.551,39.328,157.396
C00618=1038.746,76.024,-89.881,169.553,39.329,157.396
C00619=1038.752,76.273,-89.899,169.555,39.328,157.396
C00620=1038.760,76.559,-89.920,169.557,39.329,157.396
C00621=1038.767,76.845,-89.942,169.559,39.329,157.396
C00622=1038.774,77.132,-89.962,169.563,39.330,157.397
C00623=1038.781,77.418,-89.984,169.565,39.330,157.397
C00624=1038.788,77.667,-90.002,169.567,39.331,157.397
C00625=1038.794,77.915,-90.021,169.569,39.331,157.397
C00626=1038.800,78.165,-90.039,169.570,39.331,157.397
C00627=1038.806,78.414,-90.057,169.572,39.332,157.397
C00628=1038.813,78.663,-90.076,169.574,39.332,157.397
C00629=1038.819,78.913,-90.094,169.576,39.333,157.398
C00630=1038.825,79.162,-90.112,169.578,39.333,157.398
C00631=1038.831,79.412,-90.132,169.581,39.333,157.398
C00632=1038.837,79.661,-90.150,169.583,39.334,157.398
C00633=1038.844,79.910,-90.169,169.585,39.334,157.398
C00634=1038.850,80.160,-90.187,169.587,39.335,157.398
C00635=1038.856,80.408,-90.205,169.589,39.335,157.398
C00636=1038.861,80.658,-90.224,169.590,39.336,157.399
C00637=1038.868,80.907,-90.243,169.592,39.335,157.399
C00638=1038.874,81.156,-90.262,169.594,39.336,157.399
C00639=1038.881,81.405,-90.280,169.597,39.336,157.399
C00640=1038.887,81.655,-90.298,169.599,39.337,157.399
C00641=1038.893,81.904,-90.317,169.601,39.337,157.399
C00642=1038.899,82.153,-90.336,169.603,39.338,157.399
C00643=1038.905,82.402,-90.355,169.605,39.338,157.400
C00644=1038.912,82.651,-90.373,169.607,39.338,157.400
C00645=1038.918,82.901,-90.392,169.609,39.339,157.400
C00646=1038.925,83.150,-90.411,169.610,39.339,157.400
C00647=1038.930,83.399,-90.430,169.613,39.340,157.400
C00648=1038.937,83.648,-90.449,169.615,39.340,157.400
C00649=1038.943,83.898,-90.467,169.617,39.340,157.400
C00650=1038.949,84.147,-90.485,169.619,39.341,157.401
C00651=1038.956,84.396,-90.504,169.621,39.341,157.401
C00652=1038.961,84.646,-90.523,169.623,39.342,157.401
C00653=1038.968,84.895,-90.542,169.625,39.342,157.401
C00654=1038.974,85.144,-90.560,169.627,39.342,157.401
C00655=1038.981,85.393,-90.579,169.630,39.342,157.401
C00656=1038.987,85.642,-90.598,169.632,39.343,157.401
C00657=1038.993,85.892,-90.617,169.634,39.343,157.402
C00658=1038.999,86.141,-90.636,169.635,39.344,157.402
C00659=1039.006,86.390,-90.654,169.637,39.344,157.402
C00660=1039.012,86.639,-90.673,169.639,39.344,157.402
C00661=1039.018,86.888,-90.692,169.641,39.345,157.402
C00662=1039.024,87.138,-90.711,169.643,39.345,157.402
C00663=1039.031,87.387,-90.729,169.646,39.346,157.402
C00664=1039.037,87.636,-90.748,169.648,39.346,157.402
C00665=1039.043,87.885,-90.767,169.650,39.346,157.403
C00666=1039.049,88.134,-90.786,169.652,39.347,157.403
C00667=1039.055,88.383,-90.805,169.654,39.347,157.403
C00668=1039.062,88.633,-90.823,169.656,39.348,157.403
C00669=1039.068,88.882,-90.842,169.658,39.347,157.403
C00670=1039.075,89.131,-90.861,169.660,39.348,157.403
C00671=1039.080,89.380,-90.880,169.661,39.348,157.403
C00672=1039.087,89.630,-90.899,169.664,39.349,157.404
C00673=1039.094,89.879,-90.918,169.666,39.349,157.404
C00674=1039.101,90.128,-90.937,169.668,39.349,157.404
C00675=1039.106,90.377,-90.956,169.670,39.350,157.404
C00676=1039.113,90.626,-90.975,169.672,39.350,157.404
C00677=1039.118,90.876,-90.994,169.674,39.351,157.404
C00678=1039.125,91.125,-91.013,169.676,39.351,157.404
C00679=1039.131,91.374,-91.033,169.678,39.352,157.405
C00680=1039.137,91.623,-91.051,169.681,39.352,157.405
C00681=1039.143,91.872,-91.071,169.683,39.353,157.405
C00682=1039.149,92.121,-91.089,169.684,39.353,157.405
C00683=1039.155,92.371,-91.108,169.686,39.353,157.405
C00684=1039.163,92.656,-91.131,169.689,39.354,157.405
C00685=1039.170,92.943,-91.152,169.691,39.355,157.406
C00686=1039.177,93.228,-91.175,169.693,39.355,157.406
C00687=1039.184,93.515,-91.196,169.696,39.356,157.406
C00688=1039.190,93.764,-91.216,169.698,39.356,157.406
C00689=1039.197,94.013,-91.235,169.700,39.356,157.406
C00690=1039.202,94.262,-91.254,169.702,39.356,157.406
C00691=1039.209,94.511,-91.273,169.704,39.357,157.406
C00692=1039.215,94.760,-91.293,169.706,39.357,157.407
C00693=1039.221,95.009,-91.311,169.708,39.358,157.407
C00694=1039.227,95.259,-91.331,169.711,39.358,157.407
C00695=1039.234,95.508,-91.350,169.712,39.359,157.407
C00696=1039.240,95.757,-91.370,169.714,39.359,157.407
C00697=1039.246,96.007,-91.389,169.716,39.359,157.407
C00698=1039.252,96.255,-91.408,169.718,39.360,157.407
C00699=1039.258,96.505,-91.428,169.720,39.360,157.408
C00700=1039.264,96.754,-91.446,169.722,39.361,157.408
C00701=1039.271,97.003,-91.466,169.724,39.361,157.408
C00702=1039.277,97.252,-91.485,169.727,39.362,157.408
C00703=1039.283,97.502,-91.504,169.729,39.362,157.408
C00704=1039.290,97.750,-91.524,169.731,39.363,157.408
C00705=1039.296,98.000,-91.543,169.733,39.363,157.408
C00706=1039.302,98.249,-91.562,169.735,39.363,157.409
C00707=1039.309,98.498,-91.582,169.737,39.364,157.409
C00708=1039.315,98.748,-91.601,169.739,39.364,157.409
C00709=1039.321,98.996,-91.621,169.740,39.365,157.409
C00710=1039.327,99.245,-91.639,169.743,39.365,157.409
C00711=1039.333,99.494,-91.659,169.745,39.366,157.409
C00712=1039.340,99.744,-91.679,169.747,39.365,157.409
C00713=1039.346,99.994,-91.697,169.749,39.366,157.410
C00714=1039.352,100.242,-91.717,169.751,39.366,157.410
C00715=1039.359,100.491,-91.736,169.753,39.367,157.410
C00716=1039.365,100.740,-91.756,169.755,39.367,157.410
C00717=1039.371,100.990,-91.776,169.757,39.368,157.410
C00718=1039.377,101.239,-91.796,169.760,39.368,157.410
C00719=1039.384,101.488,-91.815,169.762,39.369,157.410
C00720=1039.389,101.737,-91.834,169.764,39.369,157.411
C00721=1039.395,101.986,-91.854,169.766,39.370,157.411
C00722=1039.402,102.236,-91.874,169.768,39.370,157.411
C00723=1039.408,102.485,-91.894,169.769,39.371,157.411
C00724=1039.414,102.734,-91.912,169.771,39.371,157.411
C00725=1039.420,102.983,-91.932,169.774,39.372,157.411
C00726=1039.426,103.232,-91.952,169.776,39.372,157.412
C00727=1039.432,103.482,-91.972,169.778,39.373,157.412
C00728=1039.438,103.731,-91.992,169.780,39.373,157.412
C00729=1039.445,103.979,-92.011,169.782,39.374,157.412
C00730=1039.451,104.229,-92.030,169.784,39.374,157.412
C00731=1039.457,104.478,-92.051,169.786,39.375,157.412
C00732=1039.463,104.728,-92.070,169.789,39.375,157.413
C00733=1039.469,104.976,-92.090,169.791,39.376,157.413
C00734=1039.475,105.225,-92.110,169.793,39.376,157.413
C00735=1039.482,105.475,-92.129,169.795,39.377,157.413
C00736=1039.488,105.724,-92.149,169.796,39.377,157.413
C00737=1039.494,105.973,-92.169,169.798,39.378,157.413
C00738=1039.501,106.222,-92.189,169.800,39.378,157.414
C00739=1039.506,106.472,-92.208,169.802,39.378,157.414
C00740=1039.513,106.720,-92.228,169.805,39.379,157.414
C00741=1039.519,106.969,-92.248,169.807,39.379,157.414
C00742=1039.525,107.219,-92.267,169.809,39.379,157.414
C00743=1039.531,107.468,-92.287,169.811,39.380,157.414
C00744=1039.537,107.717,-92.307,169.813,39.380,157.414
C00745=1039.544,107.966,-92.328,169.815,39.381,157.415
C00746=1039.550,108.215,-92.346,169.817,39.381,157.415
C00747=1039.556,108.464,-92.366,169.820,39.382,157.415
C00748=1039.563,108.750,-92.389,169.822,39.382,157.415
C00749=1039.571,109.036,-92.412,169.824,39.383,157.415
C00750=1039.578,109.322,-92.435,169.827,39.383,157.415
C00751=1039.585,109.608,-92.457,169.829,39.384,157.416
C00752=1039.591,109.857,-92.477,169.831,39.384,157.416
C00753=1039.598,110.107,-92.497,169.834,39.385,157.416
C00754=1039.604,110.355,-92.517,169.836,39.385,157.416
C00755=1039.610,110.604,-92.537,169.838,39.386,157.416
C00756=1039.616,110.854,-92.558,169.840,39.386,157.416
C00757=1039.622,111.103,-92.577,169.842,39.387,157.417
C00758=1039.628,111.352,-92.597,169.844,39.387,157.417
C00759=1039.635,111.601,-92.617,169.846,39.388,157.417
C00760=1039.641,111.850,-92.637,169.848,39.388,157.417
C00761=1039.647,112.100,-92.657,169.850,39.389,157.417
C00762=1039.653,112.349,-92.677,169.852,39.389,157.417
C00763=1039.659,112.597,-92.697,169.854,39.390,157.418
C00764=1039.666,112.847,-92.718,169.856,39.390,157.418
C00765=1039.672,113.096,-92.738,169.858,39.391,157.418
C00766=1039.678,113.345,-92.758,169.860,39.391,157.418
C00767=1039.684,113.594,-92.778,169.863,39.392,157.418
C00768=1039.690,113.843,-92.798,169.865,39.392,157.418
C00769=1039.696,114.092,-92.818,169.867,39.393,157.419
C00770=1039.702,114.341,-92.839,169.869,39.394,157.419
C00771=1039.708,114.590,-92.859,169.871,39.394,157.419
C00772=1039.714,114.839,-92.879,169.873,39.395,157.419
C00773=1039.720,115.089,-92.900,169.876,39.395,157.419
C00774=1039.726,115.338,-92.920,169.878,39.396,157.419
C00775=1039.732,115.587,-92.940,169.880,39.396,157.420
C00776=1039.739,115.836,-92.960,169.882,39.397,157.420
C00777=1039.744,116.085,-92.980,169.883,39.398,157.420
C00778=1039.750,116.335,-93.001,169.885,39.398,157.420
C00779=1039.756,116.584,-93.021,169.888,39.399,157.420
C00780=1039.763,116.832,-93.041,169.890,39.399,157.421
C00781=1039.769,117.082,-93.062,169.892,39.400,157.421
C00782=1039.775,117.330,-93.082,169.894,39.400,157.421
C00783=1039.781,117.580,-93.103,169.896,39.401,157.421
C00784=1039.787,117.829,-93.123,169.898,39.401,157.421
C00785=1039.792,118.078,-93.143,169.901,39.402,157.421
C00786=1039.799,118.327,-93.163,169.903,39.403,157.422
C00787=1039.805,118.576,-93.184,169.905,39.403,157.422
C00788=1039.811,118.825,-93.205,169.907,39.404,157.422
C00789=1039.817,119.074,-93.225,169.909,39.404,157.422
C00790=1039.824,119.324,-93.245,169.911,39.405,157.422
C00791=1039.830,119.572,-93.265,169.913,39.405,157.422
C00792=1039.835,119.821,-93.287,169.916,39.406,157.423
C00793=1039.842,120.071,-93.307,169.918,39.406,157.423
C00794=1039.848,120.319,-93.327,169.920,39.407,157.423
C00795=1039.854,120.569,-93.348,169.922,39.408,157.423
C00796=1039.860,120.817,-93.368,169.924,39.408,157.423
C00797=1039.867,121.067,-93.389,169.926,39.409,157.424
C00798=1039.872,121.316,-93.409,169.929,39.409,157.424
C00799=1039.879,121.565,-93.430,169.931,39.410,157.424
C00800=1039.885,121.814,-93.450,169.933,39.410,157.424
C00801=1039.891,122.063,-93.471,169.935,39.411,157.424
C00802=1039.897,122.312,-93.491,169.937,39.411,157.424
C00803=1039.903,122.562,-93.512,169.938,39.412,157.425
C00804=1039.910,122.810,-93.532,169.941,39.413,157.425
C00805=1039.915,123.060,-93.553,169.943,39.413,157.425
C00806=1039.921,123.309,-93.573,169.945,39.414,157.425
C00807=1039.928,123.558,-93.594,169.947,39.414,157.425
C00808=1039.934,123.807,-93.615,169.949,39.415,157.425
C00809=1039.940,124.056,-93.635,169.951,39.415,157.426
C00810=1039.946,124.304,-93.656,169.953,39.416,157.426
C00811=1039.952,124.554,-93.677,169.956,39.416,157.426
C00812=1039.959,124.840,-93.700,169.959,39.416,157.426
C00813=1039.967,125.126,-93.724,169.961,39.418,157.426
C00814=1039.974,125.412,-93.747,169.963,39.418,157.427
C00815=1039.981,125.697,-93.771,169.966,39.418,157.427
C00816=1039.988,125.946,-93.792,169.968,39.419,157.427
C00817=1039.994,126.196,-93.812,169.971,39.419,157.427
C00818=1039.999,126.445,-93.833,169.973,39.420,157.427
C00819=1040.006,126.694,-93.854,169.975,39.420,157.427
C00820=1040.012,126.942,-93.874,169.977,39.421,157.428
C00821=1040.018,127.192,-93.895,169.979,39.422,157.428
C00822=1040.025,127.441,-93.916,169.981,39.422,157.428
C00823=1040.031,127.689,-93.936,169.984,39.423,157.428
C00824=1040.037,127.939,-93.957,169.986,39.423,157.428
C00825=1040.043,128.187,-93.978,169.988,39.424,157.429
C00826=1040.050,128.437,-93.998,169.990,39.424,157.429
C00827=1040.056,128.687,-94.019,169.992,39.425,157.429
C00828=1040.062,128.935,-94.040,169.994,39.425,157.429
C00829=1040.068,129.185,-94.061,169.997,39.426,157.429
C00830=1040.075,129.434,-94.082,169.999,39.426,157.429
C00831=1040.081,129.682,-94.102,170.001,39.427,157.430
C00832=1040.087,129.932,-94.123,170.003,39.427,157.430
C00833=1040.093,130.180,-94.144,170.005,39.428,157.430
C00834=1040.100,130.429,-94.164,170.007,39.428,157.430
C00835=1040.106,130.678,-94.186,170.009,39.429,157.430
C00836=1040.112,130.927,-94.206,170.012,39.430,157.430
C00837=1040.118,131.177,-94.228,170.014,39.430,157.431
C00838=1040.125,131.426,-94.248,170.016,39.431,157.431
C00839=1040.131,131.675,-94.269,170.018,39.431,157.431
C00840=1040.137,131.924,-94.291,170.020,39.432,157.431
C00841=1040.143,132.173,-94.311,170.023,39.433,157.431
C00842=1040.149,132.422,-94.333,170.025,39.433,157.432
C00843=1040.156,132.671,-94.354,170.027,39.434,157.432
C00844=1040.162,132.920,-94.374,170.029,39.434,157.432
C00845=1040.167,133.169,-94.396,170.031,39.435,157.432
C00846=1040.174,133.418,-94.417,170.034,39.436,157.432
C00847=1040.180,133.667,-94.438,170.037,39.436,157.433
C00848=1040.185,133.916,-94.459,170.039,39.437,157.433
C00849=1040.192,134.165,-94.480,170.041,39.437,157.433
C00850=1040.199,134.414,-94.502,170.043,39.438,157.433
C00851=1040.204,134.663,-94.523,170.045,39.439,157.433
C00852=1040.211,134.912,-94.543,170.047,39.439,157.434
C00853=1040.217,135.162,-94.565,170.050,39.440,157.434
C00854=1040.222,135.410,-94.586,170.052,39.440,157.434
C00855=1040.229,135.659,-94.607,170.054,39.441,157.434
C00856=1040.235,135.909,-94.628,170.056,39.442,157.434
C00857=1040.241,136.157,-94.649,170.058,39.442,157.434
C00858=1040.248,136.406,-94.670,170.060,39.443,157.435
C00859=1040.254,136.655,-94.692,170.063,39.443,157.435
C00860=1040.260,136.905,-94.714,170.065,39.444,157.435
C00861=1040.266,137.153,-94.735,170.067,39.445,157.435
C00862=1040.272,137.403,-94.755,170.069,39.445,157.435
C00863=1040.278,137.652,-94.777,170.071,39.446,157.436
C00864=1040.284,137.900,-94.798,170.074,39.447,157.436
C00865=1040.290,138.149,-94.820,170.076,39.447,157.436
C00866=1040.297,138.398,-94.841,170.078,39.448,157.436
C00867=1040.303,138.648,-94.863,170.081,39.448,157.436
C00868=1040.309,138.896,-94.884,170.083,39.449,157.437
C00869=1040.315,139.145,-94.905,170.085,39.450,157.437
C00870=1040.322,139.394,-94.926,170.088,39.450,157.437
C00871=1040.328,139.644,-94.947,170.090,39.451,157.437
C00872=1040.333,139.893,-94.969,170.092,39.452,157.437
C00873=1040.339,140.142,-94.990,170.094,39.452,157.438
C00874=1040.345,140.391,-95.012,170.096,39.453,157.438
C00875=1040.352,140.640,-95.034,170.099,39.454,157.438
C00876=1040.358,140.925,-95.059,170.101,39.454,157.438
C00877=1040.366,141.211,-95.083,170.104,39.455,157.439
C00878=1040.372,141.496,-95.108,170.106,39.456,157.439
C00879=1040.380,141.782,-95.133,170.108,39.457,157.439
C00880=1040.385,142.031,-95.154,170.112,39.457,157.439
C00881=1040.391,142.280,-95.176,170.114,39.458,157.439
C00882=1040.397,142.529,-95.197,170.116,39.459,157.440
C00883=1040.404,142.778,-95.218,170.118,39.459,157.440
C00884=1040.411,143.027,-95.240,170.120,39.460,157.440
C00885=1040.416,143.276,-95.261,170.123,39.461,157.440
C00886=1040.422,143.525,-95.283,170.125,39.461,157.440
C00887=1040.428,143.774,-95.305,170.127,39.462,157.441
C00888=1040.435,144.023,-95.327,170.129,39.463,157.441
C00889=1040.441,144.272,-95.349,170.131,39.463,157.441
C00890=1040.447,144.520,-95.370,170.133,39.464,157.441
C00891=1040.453,144.770,-95.391,170.136,39.465,157.442
C00892=1040.459,145.019,-95.413,170.139,39.465,157.442
C00893=1040.465,145.268,-95.435,170.141,39.466,157.442
C00894=1040.471,145.517,-95.456,170.143,39.466,157.442
C00895=1040.478,145.766,-95.479,170.145,39.467,157.442
C00896=1040.484,146.015,-95.500,170.148,39.468,157.442
C00897=1040.489,146.264,-95.522,170.150,39.468,157.443
C00898=1040.496,146.513,-95.543,170.152,39.470,157.443
C00899=1040.502,146.762,-95.565,170.154,39.470,157.443
C00900=1040.508,147.011,-95.587,170.156,39.470,157.443
C00901=1040.514,147.260,-95.609,170.159,39.472,157.444
C00902=1040.521,147.509,-95.631,170.162,39.472,157.444
C00903=1040.527,147.758,-95.652,170.164,39.473,157.444
C00904=1040.533,148.007,-95.675,170.166,39.474,157.444
C00905=1040.539,148.255,-95.696,170.168,39.474,157.444
C00906=1040.545,148.504,-95.717,170.171,39.475,157.445
C00907=1040.551,148.753,-95.740,170.173,39.476,157.445
C00908=1040.558,149.002,-95.761,170.175,39.477,157.445
C00909=1040.563,149.252,-95.784,170.177,39.477,157.445
C00910=1040.569,149.500,-95.806,170.179,39.478,157.445
C00911=1040.576,149.750,-95.828,170.183,39.479,157.446
C00912=1040.582,149.999,-95.849,170.185,39.479,157.446
C00913=1040.588,150.247,-95.871,170.187,39.480,157.446
C00914=1040.594,150.496,-95.893,170.189,39.481,157.446
C00915=1040.599,150.745,-95.915,170.192,39.482,157.447
C00916=1040.606,150.994,-95.937,170.194,39.482,157.447
C00917=1040.612,151.243,-95.959,170.196,39.483,157.447
C00918=1040.618,151.492,-95.981,170.198,39.484,157.447
C00919=1040.624,151.741,-96.004,170.201,39.484,157.448
C00920=1040.630,151.990,-96.026,170.204,39.485,157.448
C00921=1040.636,152.239,-96.048,170.206,39.486,157.448
C00922=1040.643,152.488,-96.069,170.208,39.487,157.448
C00923=1040.649,152.737,-96.092,170.210,39.487,157.448
C00924=1040.654,152.986,-96.114,170.212,39.488,157.449
C00925=1040.661,153.235,-96.136,170.215,39.489,157.449
C00926=1040.667,153.484,-96.158,170.218,39.489,157.449
C00927=1040.674,153.733,-96.180,170.220,39.490,157.449
C00928=1040.680,153.982,-96.202,170.222,39.491,157.450
C00929=1040.685,154.231,-96.225,170.224,39.492,157.450
C00930=1040.692,154.480,-96.246,170.227,39.492,157.450
C00931=1040.698,154.729,-96.269,170.229,39.494,157.450
C00932=1040.703,154.977,-96.291,170.231,39.494,157.450
C00933=1040.709,155.226,-96.313,170.234,39.495,157.451
C00934=1040.716,155.475,-96.335,170.236,39.496,157.451
C00935=1040.721,155.724,-96.358,170.239,39.497,157.451
C00936=1040.728,155.973,-96.380,170.241,39.497,157.451
C00937=1040.734,156.221,-96.402,170.243,39.498,157.452
C00938=1040.740,156.471,-96.425,170.245,39.499,157.452
C00939=1040.746,156.719,-96.447,170.249,39.500,157.452
C00940=1040.753,157.005,-96.472,170.251,39.500,157.452
C00941=1040.761,157.290,-96.498,170.253,39.501,157.453
C00942=1040.767,157.576,-96.524,170.256,39.502,157.453
C00943=1040.774,157.861,-96.550,170.259,39.503,157.453
C00944=1040.780,158.110,-96.572,170.262,39.504,157.453
C00945=1040.787,158.359,-96.594,170.264,39.505,157.454
C00946=1040.792,158.608,-96.617,170.266,39.505,157.454
C00947=1040.799,158.856,-96.639,170.268,39.506,157.454
C00948=1040.804,159.106,-96.661,170.271,39.507,157.454
C00949=1040.811,159.354,-96.684,170.274,39.508,157.455
C00950=1040.817,159.603,-96.706,170.276,39.508,157.455
C00951=1040.823,159.852,-96.728,170.278,39.509,157.455
C00952=1040.829,160.101,-96.751,170.280,39.510,157.455
C00953=1040.835,160.351,-96.774,170.283,39.511,157.456
C00954=1040.842,160.599,-96.796,170.285,39.512,157.456
C00955=1040.848,160.848,-96.819,170.288,39.513,157.456
C00956=1040.853,161.097,-96.842,170.290,39.514,157.456
C00957=1040.859,161.346,-96.865,170.293,39.515,157.457
C00958=1040.865,161.595,-96.887,170.295,39.516,157.457
C00959=1040.871,161.844,-96.910,170.297,39.516,157.457
C00960=1040.877,162.093,-96.933,170.299,39.517,157.457
C00961=1040.882,162.342,-96.956,170.303,39.518,157.458
C00962=1040.888,162.591,-96.979,170.305,39.519,157.458
C00963=1040.895,162.839,-97.001,170.307,39.520,157.458
C00964=1040.900,163.088,-97.024,170.309,39.521,157.458
C00965=1040.906,163.337,-97.047,170.312,39.522,157.459
C00966=1040.912,163.586,-97.070,170.314,39.523,157.459
C00967=1040.918,163.835,-97.093,170.317,39.524,157.459
C00968=1040.924,164.083,-97.115,170.319,39.525,157.460
C00969=1040.930,164.332,-97.138,170.322,39.526,157.460
C00970=1040.936,164.581,-97.161,170.324,39.527,157.460
C00971=1040.941,164.830,-97.184,170.326,39.527,157.460
C00972=1040.947,165.079,-97.207,170.329,39.528,157.461
C00973=1040.954,165.328,-97.230,170.332,39.529,157.461
C00974=1040.960,165.577,-97.253,170.334,39.531,157.461
C00975=1040.966,165.826,-97.275,170.336,39.531,157.461
C00976=1040.971,166.075,-97.298,170.338,39.532,157.462
C00977=1040.977,166.323,-97.322,170.342,39.533,157.462
C00978=1040.984,166.572,-97.344,170.344,39.534,157.462
C00979=1040.990,166.821,-97.367,170.346,39.535,157.462
C00980=1040.995,167.070,-97.390,170.348,39.536,157.463
C00981=1041.002,167.319,-97.414,170.351,39.537,157.463
C00982=1041.007,167.568,-97.437,170.354,39.538,157.463
C00983=1041.013,167.817,-97.460,170.356,39.538,157.464
C00984=1041.020,168.066,-97.482,170.358,39.539,157.464
C00985=1041.026,168.314,-97.506,170.361,39.541,157.464
C00986=1041.031,168.563,-97.528,170.364,39.542,157.464
C00987=1041.038,168.812,-97.552,170.366,39.542,157.465
C00988=1041.043,169.061,-97.575,170.368,39.543,157.465
C00989=1041.050,169.310,-97.597,170.371,39.544,157.465
C00990=1041.056,169.559,-97.620,170.374,39.545,157.465
C00991=1041.062,169.807,-97.644,170.376,39.546,157.466
C00992=1041.068,170.057,-97.667,170.378,39.547,157.466
C00993=1041.074,170.306,-97.690,170.381,39.548,157.466
C00994=1041.079,170.554,-97.713,170.384,39.549,157.467
C00995=1041.085,170.803,-97.737,170.386,39.550,157.467
C00996=1041.092,171.052,-97.759,170.388,39.550,157.467
C00997=1041.098,171.301,-97.782,170.391,39.552,157.467
C00998=1041.104,171.550,-97.805,170.394,39.553,157.468
C00999=1041.110,171.798,-97.829,170.396,39.554,157.468
C01000=1041.116,172.048,-97.852,170.399,39.554,157.468
C01001=1041.122,172.297,-97.875,170.401,39.555,157.468
C01002=1041.129,172.544,-97.898,170.404,39.556,157.469
C01003=1041.135,172.793,-97.921,170.406,39.557,157.469
C01004=1041.141,173.079,-97.948,170.410,39.558,157.469
C01005=1041.149,173.363,-97.974,170.412,39.559,157.470
C01006=1041.155,173.648,-98.001,170.415,39.560,157.470
C01007=1041.162,173.933,-98.028,170.418,39.561,157.470
C01008=1041.169,174.182,-98.050,170.421,39.562,157.471
C01009=1041.175,174.431,-98.075,170.423,39.564,157.471
C01010=1041.181,174.679,-98.097,170.425,39.564,157.471
C01011=1041.187,174.928,-98.120,170.429,39.565,157.471
C01012=1041.193,175.177,-98.144,170.431,39.566,157.472
C01013=1041.199,175.426,-98.167,170.433,39.567,157.472
C01014=1041.205,175.675,-98.191,170.436,39.568,157.472
C01015=1041.212,175.924,-98.214,170.439,39.569,157.472
C01016=1041.218,176.173,-98.237,170.441,39.570,157.473
C01017=1041.224,176.421,-98.260,170.444,39.571,157.473
C01018=1041.230,176.671,-98.284,170.446,39.572,157.473
C01019=1041.236,176.919,-98.307,170.449,39.573,157.474
C01020=1041.243,177.168,-98.331,170.452,39.573,157.474
C01021=1041.249,177.417,-98.354,170.454,39.574,157.474
C01022=1041.255,177.666,-98.377,170.456,39.575,157.474
C01023=1041.261,177.915,-98.401,170.460,39.576,157.475
C01024=1041.267,178.164,-98.424,170.462,39.578,157.475
C01025=1041.274,178.412,-98.448,170.464,39.578,157.475
C01026=1041.280,178.660,-98.471,170.467,39.579,157.476
C01027=1041.286,178.909,-98.494,170.470,39.580,157.476
C01028=1041.293,179.158,-98.518,170.472,39.581,157.476
C01029=1041.298,179.407,-98.541,170.475,39.582,157.476
C01030=1041.305,179.656,-98.565,170.478,39.583,157.477
C01031=1041.311,179.905,-98.588,170.481,39.584,157.477
C01032=1041.317,180.154,-98.612,170.483,39.585,157.477
C01033=1041.323,180.402,-98.636,170.485,39.586,157.477
C01034=1041.330,180.652,-98.659,170.489,39.587,157.478
C01035=1041.337,180.900,-98.682,170.491,39.588,157.478
C01036=1041.343,181.149,-98.706,170.493,39.589,157.478
C01037=1041.349,181.398,-98.729,170.496,39.589,157.479
C01038=1041.356,181.647,-98.753,170.499,39.590,157.479
C01039=1041.362,181.895,-98.777,170.502,39.591,157.479
C01040=1041.368,182.145,-98.800,170.504,39.593,157.480
C01041=1041.374,182.393,-98.824,170.507,39.594,157.480
C01042=1041.381,182.642,-98.848,170.510,39.595,157.480
C01043=1041.386,182.891,-98.871,170.512,39.596,157.480
C01044=1041.393,183.140,-98.895,170.515,39.596,157.481
C01045=1041.399,183.388,-98.919,170.518,39.597,157.481
C01046=1041.406,183.637,-98.943,170.520,39.598,157.481
C01047=1041.411,183.886,-98.966,170.523,39.599,157.482
C01048=1041.417,184.135,-98.990,170.525,39.600,157.482
C01049=1041.423,184.384,-99.014,170.529,39.602,157.482
C01050=1041.429,184.632,-99.038,170.531,39.603,157.483
C01051=1041.435,184.881,-99.062,170.533,39.604,157.483
C01052=1041.441,185.130,-99.086,170.537,39.605,157.483
C01053=1041.447,185.379,-99.110,170.539,39.606,157.483
C01054=1041.453,185.627,-99.135,170.541,39.607,157.484
C01055=1041.459,185.876,-99.159,170.545,39.609,157.484
C01056=1041.465,186.124,-99.182,170.547,39.610,157.485
C01057=1041.471,186.374,-99.207,170.549,39.611,157.485
C01058=1041.477,186.622,-99.231,170.553,39.612,157.485
C01059=1041.483,186.871,-99.255,170.555,39.613,157.485
C01060=1041.489,187.120,-99.279,170.558,39.615,157.486
C01061=1041.495,187.369,-99.304,170.561,39.616,157.486
C01062=1041.501,187.617,-99.327,170.563,39.617,157.486
C01063=1041.507,187.866,-99.352,170.566,39.618,157.487
C01064=1041.513,188.115,-99.375,170.568,39.619,157.487
C01065=1041.519,188.364,-99.400,170.572,39.621,157.488
C01066=1041.525,188.612,-99.424,170.574,39.622,157.488
C01067=1041.531,188.861,-99.449,170.576,39.623,157.488
C01068=1041.538,189.146,-99.476,170.580,39.624,157.488
C01069=1041.545,189.429,-99.504,170.583,39.625,157.489
C01070=1041.552,189.714,-99.532,170.587,39.627,157.489
C01071=1041.559,189.999,-99.560,170.589,39.628,157.490
C01072=1041.565,190.247,-99.584,170.592,39.629,157.490
C01073=1041.571,190.496,-99.608,170.595,39.631,157.490
C01074=1041.577,190.745,-99.632,170.598,39.632,157.491
C01075=1041.582,190.994,-99.657,170.600,39.633,157.491
C01076=1041.589,191.243,-99.681,170.604,39.634,157.491
C01077=1041.595,191.491,-99.706,170.606,39.635,157.492
C01078=1041.601,191.740,-99.730,170.608,39.637,157.492
C01079=1041.607,191.989,-99.754,170.612,39.638,157.492
C01080=1041.613,192.237,-99.778,170.614,39.639,157.493
C01081=1041.619,192.486,-99.803,170.617,39.640,157.493
C01082=1041.626,192.734,-99.827,170.620,39.641,157.493
C01083=1041.631,192.984,-99.852,170.623,39.642,157.494
C01084=1041.638,193.233,-99.876,170.625,39.644,157.494
C01085=1041.644,193.481,-99.901,170.628,39.645,157.494
C01086=1041.650,193.730,-99.925,170.631,39.646,157.495
C01087=1041.656,193.979,-99.949,170.634,39.647,157.495
C01088=1041.662,194.227,-99.974,170.636,39.648,157.495
C01089=1041.668,194.476,-99.998,170.640,39.650,157.496
C01090=1041.674,194.725,-100.023,170.642,39.651,157.496
C01091=1041.681,194.973,-100.048,170.645,39.652,157.497
C01092=1041.687,195.222,-100.072,170.648,39.653,157.497
C01093=1041.693,195.471,-100.096,170.651,39.655,157.497
C01094=1041.699,195.720,-100.121,170.653,39.656,157.498
C01095=1041.705,195.968,-100.145,170.657,39.657,157.498
C01096=1041.712,196.217,-100.170,170.659,39.658,157.498
C01097=1041.718,196.466,-100.195,170.662,39.659,157.499
C01098=1041.724,196.715,-100.219,170.665,39.660,157.499
C01099=1041.730,196.963,-100.244,170.668,39.661,157.499
C01100=1041.736,197.212,-100.268,170.670,39.663,157.500
C01101=1041.743,197.460,-100.293,170.674,39.664,157.500
C01102=1041.749,197.709,-100.317,170.676,39.665,157.500
C01103=1041.755,197.957,-100.342,170.680,39.667,157.501
C01104=1041.761,198.207,-100.367,170.682,39.668,157.501
C01105=1041.768,198.455,-100.392,170.685,39.669,157.501
C01106=1041.774,198.704,-100.416,170.688,39.671,157.502
C01107=1041.781,198.953,-100.441,170.691,39.672,157.502
C01108=1041.786,199.201,-100.465,170.693,39.673,157.502
C01109=1041.793,199.450,-100.490,170.697,39.674,157.503
C01110=1041.799,199.699,-100.515,170.699,39.675,157.503
C01111=1041.805,199.948,-100.540,170.702,39.676,157.503
C01112=1041.812,200.196,-100.565,170.706,39.678,157.504
C01113=1041.818,200.445,-100.589,170.708,39.679,157.504
C01114=1041.825,200.694,-100.614,170.711,39.680,157.505
C01115=1041.830,200.942,-100.638,170.714,39.682,157.505
C01116=1041.836,201.191,-100.664,170.717,39.683,157.505
C01117=1041.842,201.440,-100.689,170.719,39.684,157.506
C01118=1041.848,201.689,-100.714,170.723,39.685,157.506
C01119=1041.855,201.937,-100.738,170.725,39.687,157.507
C01120=1041.861,202.186,-100.764,170.728,39.688,157.507
C01121=1041.867,202.434,-100.789,170.732,39.690,157.507
C01122=1041.873,202.682,-100.814,170.734,39.691,157.508
C01123=1041.879,202.932,-100.839,170.738,39.692,157.508
C01124=1041.885,203.180,-100.864,170.740,39.694,157.508
C01125=1041.892,203.429,-100.889,170.743,39.695,157.509
C01126=1041.898,203.678,-100.915,170.746,39.697,157.509
C01127=1041.904,203.926,-100.940,170.749,39.698,157.510
C01128=1041.909,204.175,-100.964,170.751,39.699,157.510
C01129=1041.916,204.424,-100.990,170.755,39.701,157.510
C01130=1041.922,204.672,-101.015,170.758,39.702,157.511
C01131=1041.928,204.921,-101.040,170.761,39.704,157.511
C01132=1041.954,205.972,-101.147,171.038,39.806,157.543
C01133=1041.962,206.268,-101.178,171.040,39.808,157.543
C01134=1041.970,206.564,-101.209,171.043,39.811,157.544
C01135=1041.979,206.860,-101.241,171.045,39.814,157.544
C01136=1041.987,207.156,-101.272,171.048,39.817,157.545
C01137=1041.992,207.405,-101.298,171.051,39.818,157.546
C01138=1042.000,207.653,-101.325,171.052,39.821,157.546
C01139=1042.006,207.901,-101.351,171.055,39.823,157.547
C01140=1042.013,208.150,-101.377,171.057,39.825,157.547
C01141=1042.019,208.399,-101.404,171.059,39.827,157.548
C01142=1042.026,208.647,-101.430,171.061,39.829,157.548
C01143=1042.033,208.896,-101.457,171.064,39.831,157.549
C01144=1042.039,209.144,-101.483,171.065,39.833,157.549
C01145=1042.046,209.393,-101.510,171.068,39.836,157.550
C01146=1042.053,209.641,-101.537,171.071,39.838,157.550
C01147=1042.059,209.890,-101.564,171.072,39.840,157.551
C01148=1042.066,210.138,-101.590,171.075,39.842,157.551
C01149=1042.073,210.386,-101.616,171.077,39.844,157.552
C01150=1042.079,210.636,-101.643,171.079,39.847,157.553
C01151=1042.086,210.884,-101.669,171.081,39.848,157.553
C01152=1042.092,211.133,-101.696,171.084,39.850,157.554
C01153=1042.099,211.381,-101.722,171.085,39.853,157.554
C01154=1042.106,211.629,-101.749,171.088,39.855,157.555
C01155=1042.112,211.878,-101.776,171.090,39.857,157.555
C01156=1042.119,212.126,-101.802,171.092,39.859,157.556
C01157=1042.125,212.375,-101.829,171.095,39.861,157.556
C01158=1042.131,212.623,-101.857,171.097,39.863,157.557
C01159=1042.139,212.872,-101.883,171.099,39.866,157.557
C01160=1042.145,213.121,-101.910,171.101,39.868,157.558
C01161=1042.151,213.369,-101.936,171.104,39.870,157.558
C01162=1042.158,213.617,-101.964,171.105,39.872,157.559
C01163=1042.165,213.866,-101.990,171.108,39.874,157.559
C01164=1042.171,214.114,-102.017,171.110,39.876,157.560
C01165=1042.178,214.362,-102.044,171.112,39.879,157.561
C01166=1042.184,214.611,-102.071,171.114,39.880,157.561
C01167=1042.191,214.860,-102.098,171.117,39.883,157.562
C01168=1042.198,215.108,-102.125,171.120,39.885,157.562
C01169=1042.204,215.356,-102.152,171.121,39.887,157.563
C01170=1042.211,215.605,-102.178,171.124,39.889,157.563
C01171=1042.218,215.853,-102.206,171.126,39.891,157.564
C01172=1042.224,216.101,-102.232,171.128,39.894,157.564
C01173=1042.230,216.351,-102.259,171.130,39.895,157.565
C01174=1042.237,216.599,-102.287,171.133,39.898,157.565
C01175=1042.244,216.848,-102.313,171.135,39.900,157.566
C01176=1042.250,217.095,-102.340,171.137,39.902,157.566
C01177=1042.257,217.344,-102.367,171.139,39.904,157.567
C01178=1042.264,217.593,-102.394,171.142,39.906,157.567
C01179=1042.271,217.841,-102.421,171.144,39.908,157.568
C01180=1042.277,218.090,-102.448,171.146,39.910,157.568
C01181=1042.284,218.338,-102.475,171.149,39.913,157.569
C01182=1042.291,218.587,-102.502,171.151,39.914,157.569
C01183=1042.297,218.835,-102.529,171.154,39.916,157.570
C01184=1042.304,219.083,-102.556,171.155,39.919,157.571
C01185=1042.311,219.332,-102.583,171.158,39.920,157.571
C01186=1042.317,219.581,-102.610,171.160,39.923,157.572
C01187=1042.324,219.828,-102.637,171.163,39.925,157.572
C01188=1042.330,220.077,-102.664,171.165,39.927,157.573
C01189=1042.339,220.379,-102.697,171.168,39.930,157.573
C01190=1042.346,220.680,-102.730,171.171,39.932,157.574
C01191=1042.354,220.982,-102.764,171.173,39.935,157.575
C01192=1042.362,221.283,-102.797,171.176,39.938,157.575
C01193=1042.369,221.532,-102.824,171.179,39.939,157.576
C01194=1042.376,221.780,-102.851,171.181,39.942,157.576
C01195=1042.382,222.028,-102.878,171.183,39.944,157.577
C01196=1042.389,222.277,-102.906,171.185,39.946,157.578
C01197=1042.395,222.526,-102.933,171.188,39.948,157.578
C01198=1042.402,222.774,-102.961,171.190,39.950,157.579
C01199=1042.408,223.022,-102.988,171.193,39.952,157.579
C01200=1042.414,223.271,-103.015,171.194,39.955,157.580
C01201=1042.422,223.519,-103.042,171.197,39.956,157.580
C01202=1042.428,223.768,-103.070,171.200,39.959,157.581
C01203=1042.435,224.016,-103.098,171.202,39.961,157.581
C01204=1042.441,224.264,-103.124,171.205,39.963,157.582
C01205=1042.447,224.513,-103.152,171.206,39.965,157.582
C01206=1042.454,224.761,-103.180,171.209,39.967,157.583
C01207=1042.461,225.010,-103.207,171.211,39.970,157.583
C01208=1042.468,225.258,-103.235,171.214,39.971,157.584
C01209=1042.475,225.507,-103.262,171.216,39.973,157.584
C01210=1042.481,225.755,-103.289,171.219,39.976,157.585
C01211=1042.487,226.003,-103.317,171.222,39.978,157.586
C01212=1042.494,226.251,-103.344,171.223,39.980,157.586
C01213=1042.501,226.500,-103.372,171.226,39.982,157.587
C01214=1042.507,226.749,-103.399,171.228,39.984,157.587
C01215=1042.514,226.997,-103.427,171.231,39.986,157.588
C01216=1042.521,227.246,-103.454,171.233,39.988,157.588
C01217=1042.528,227.494,-103.482,171.236,39.990,157.589
C01218=1042.535,227.742,-103.509,171.238,39.992,157.589
C01219=1042.541,227.990,-103.537,171.240,39.994,157.590
C01220=1042.547,228.239,-103.565,171.243,39.997,157.590
C01221=1042.554,228.487,-103.592,171.245,39.999,157.591
C01222=1042.561,228.735,-103.620,171.248,40.001,157.591
C01223=1042.567,228.984,-103.648,171.250,40.003,157.592
C01224=1042.574,229.232,-103.675,171.253,40.005,157.593
C01225=1042.581,229.481,-103.703,171.255,40.007,157.593
C01226=1042.587,229.729,-103.731,171.258,40.009,157.594
C01227=1042.594,229.978,-103.759,171.259,40.011,157.594
C01228=1042.600,230.226,-103.787,171.262,40.014,157.595
C01229=1042.606,230.474,-103.814,171.265,40.016,157.595
C01230=1042.613,230.723,-103.842,171.267,40.018,157.596
C01231=1042.619,230.971,-103.870,171.270,40.020,157.596
C01232=1042.626,231.219,-103.898,171.272,40.022,157.597
C01233=1042.633,231.468,-103.925,171.275,40.024,157.598
C01234=1042.640,231.716,-103.953,171.277,40.026,157.598
C01235=1042.646,231.965,-103.981,171.280,40.028,157.599
C01236=1042.652,232.213,-104.010,171.282,40.031,157.599
C01237=1042.659,232.461,-104.037,171.284,40.033,157.600
C01238=1042.666,232.710,-104.065,171.287,40.035,157.600
C01239=1042.673,232.958,-104.093,171.289,40.037,157.601
C01240=1042.678,233.207,-104.121,171.292,40.039,157.601
C01241=1042.685,233.455,-104.150,171.294,40.041,157.602
C01242=1042.692,233.703,-104.177,171.297,40.044,157.603
C01243=1042.699,233.952,-104.205,171.300,40.046,157.603
C01244=1042.705,234.200,-104.234,171.302,40.048,157.604
C01245=1042.713,234.494,-104.266,171.305,40.050,157.604
C01246=1042.721,234.788,-104.300,171.307,40.053,157.605
C01247=1042.728,235.082,-104.333,171.311,40.055,157.606
C01248=1042.736,235.376,-104.366,171.314,40.058,157.606
C01249=1042.743,235.624,-104.394,171.316,40.060,157.607
C01250=1042.749,235.872,-104.423,171.319,40.062,157.607
C01251=1042.756,236.121,-104.451,171.322,40.064,157.608
C01252=1042.762,236.369,-104.478,171.324,40.066,157.608
C01253=1042.769,236.617,-104.507,171.327,40.068,157.609
C01254=1042.775,236.866,-104.535,171.329,40.071,157.610
C01255=1042.782,237.114,-104.563,171.332,40.073,157.610
C01256=1042.789,237.362,-104.591,171.334,40.075,157.611
C01257=1042.795,237.611,-104.620,171.337,40.077,157.611
C01258=1042.802,237.860,-104.648,171.340,40.079,157.612
C01259=1042.809,238.108,-104.676,171.342,40.081,157.612
C01260=1042.816,238.356,-104.704,171.345,40.084,157.613
C01261=1042.822,238.605,-104.733,171.347,40.085,157.613
C01262=1042.829,238.853,-104.761,171.350,40.087,157.614
C01263=1042.835,239.101,-104.790,171.352,40.090,157.615
C01264=1042.842,239.350,-104.818,171.355,40.092,157.615
C01265=1042.849,239.597,-104.846,171.358,40.094,157.616
C01266=1042.855,239.846,-104.874,171.360,40.096,157.616
C01267=1042.862,240.094,-104.903,171.363,40.098,157.617
C01268=1042.868,240.342,-104.931,171.365,40.100,157.617
C01269=1042.875,240.591,-104.960,171.368,40.103,157.618
C01270=1042.882,240.840,-104.988,171.370,40.104,157.618
C01271=1042.889,241.087,-105.016,171.373,40.106,157.619
C01272=1042.895,241.336,-105.044,171.376,40.109,157.620
C01273=1042.902,241.584,-105.073,171.378,40.111,157.620
C01274=1042.908,241.832,-105.102,171.381,40.113,157.621
C01275=1042.914,242.081,-105.130,171.383,40.115,157.621
C01276=1042.921,242.329,-105.159,171.386,40.118,157.622
C01277=1042.927,242.577,-105.188,171.388,40.119,157.622
C01278=1042.934,242.826,-105.216,171.391,40.122,157.623
C01279=1042.941,243.074,-105.245,171.394,40.124,157.623
C01280=1042.947,243.322,-105.274,171.396,40.126,157.624
C01281=1042.954,243.571,-105.302,171.399,40.128,157.625
C01282=1042.960,243.819,-105.331,171.402,40.131,157.625
C01283=1042.967,244.067,-105.359,171.404,40.133,157.626
C01284=1042.973,244.315,-105.388,171.407,40.134,157.626
C01285=1042.980,244.564,-105.417,171.409,40.137,157.627
C01286=1042.987,244.812,-105.445,171.412,40.139,157.627
C01287=1042.993,245.060,-105.474,171.414,40.141,157.628
C01288=1043.000,245.308,-105.503,171.417,40.143,157.629
C01289=1043.006,245.557,-105.531,171.420,40.146,157.629
C01290=1043.012,245.805,-105.560,171.422,40.148,157.630
C01291=1043.019,246.054,-105.590,171.426,40.150,157.630
C01292=1043.025,246.302,-105.619,171.429,40.152,157.631
C01293=1043.031,246.550,-105.648,171.431,40.155,157.632
C01294=1043.038,246.798,-105.677,171.434,40.157,157.632
C01295=1043.045,247.046,-105.705,171.436,40.159,157.633
C01296=1043.051,247.294,-105.734,171.439,40.161,157.633
C01297=1043.058,247.543,-105.764,171.442,40.164,157.634
C01298=1043.064,247.791,-105.793,171.444,40.165,157.634
C01299=1043.070,248.039,-105.822,171.447,40.167,157.635
C01300=1043.076,248.287,-105.851,171.449,40.170,157.636
C01301=1043.084,248.576,-105.884,171.453,40.172,157.636
C01302=1043.091,248.864,-105.918,171.456,40.175,157.637
C01303=1043.099,249.152,-105.952,171.458,40.178,157.638
C01304=1043.106,249.440,-105.985,171.462,40.180,157.638
C01305=1043.113,249.688,-106.014,171.465,40.183,157.639
C01306=1043.120,249.937,-106.043,171.467,40.185,157.640
C01307=1043.126,250.185,-106.072,171.470,40.187,157.640
C01308=1043.133,250.433,-106.101,171.473,40.189,157.641
C01309=1043.139,250.681,-106.131,171.475,40.191,157.641
C01310=1043.146,250.930,-106.160,171.479,40.193,157.642
C01311=1043.152,251.178,-106.189,171.481,40.195,157.642
C01312=1043.159,251.426,-106.218,171.484,40.197,157.643
C01313=1043.166,251.675,-106.248,171.487,40.200,157.644
C01314=1043.172,251.923,-106.276,171.489,40.202,157.644
C01315=1043.179,252.171,-106.305,171.492,40.204,157.645
C01316=1043.185,252.419,-106.334,171.494,40.206,157.645
C01317=1043.192,252.667,-106.365,171.498,40.209,157.646
C01318=1043.198,252.915,-106.394,171.501,40.211,157.647
C01319=1043.205,253.163,-106.423,171.503,40.213,157.647
C01320=1043.211,253.412,-106.452,171.506,40.215,157.648
C01321=1043.218,253.660,-106.482,171.509,40.218,157.648
C01322=1043.225,253.908,-106.511,171.511,40.220,157.649
C01323=1043.231,254.157,-106.540,171.515,40.222,157.650
C01324=1043.237,254.405,-106.569,171.517,40.224,157.650
C01325=1043.245,254.653,-106.599,171.520,40.226,157.651
C01326=1043.252,254.901,-106.628,171.523,40.228,157.651
C01327=1043.258,255.149,-106.657,171.525,40.230,157.652
C01328=1043.265,255.398,-106.686,171.529,40.232,157.652
C01329=1043.271,255.645,-106.716,171.531,40.235,157.653
C01330=1043.278,255.894,-106.745,171.534,40.237,157.654
C01331=1043.284,256.142,-106.774,171.537,40.239,157.654
C01332=1043.291,256.390,-106.804,171.539,40.241,157.655
C01333=1043.298,256.639,-106.834,171.543,40.243,157.655
C01334=1043.304,256.886,-106.863,171.546,40.246,157.656
C01335=1043.311,257.135,-106.893,171.548,40.248,157.657
C01336=1043.317,257.383,-106.922,171.551,40.250,157.657
C01337=1043.325,257.631,-106.952,171.554,40.252,157.658
C01338=1043.332,257.879,-106.980,171.557,40.254,157.658
C01339=1043.339,258.127,-107.011,171.560,40.257,157.659
C01340=1043.345,258.375,-107.040,171.562,40.259,157.660
C01341=1043.352,258.624,-107.069,171.566,40.260,157.660
C01342=1043.358,258.872,-107.099,171.568,40.263,157.661
C01343=1043.365,259.121,-107.128,171.571,40.265,157.661
C01344=1043.372,259.368,-107.158,171.574,40.267,157.662
C01345=1043.379,259.617,-107.187,171.577,40.269,157.662
C01346=1043.385,259.864,-107.217,171.580,40.271,157.663
C01347=1043.392,260.113,-107.246,171.583,40.274,157.664
C01348=1043.399,260.361,-107.276,171.586,40.276,157.664
C01349=1043.406,260.609,-107.306,171.589,40.278,157.665
C01350=1043.412,260.857,-107.335,171.591,40.280,157.665
C01351=1043.419,261.105,-107.366,171.594,40.282,157.666
C01352=1043.425,261.353,-107.395,171.598,40.285,157.667
C01353=1043.433,261.602,-107.425,171.600,40.287,157.667
C01354=1043.439,261.850,-107.454,171.603,40.289,157.668
C01355=1043.446,262.098,-107.484,171.606,40.291,157.668
C01356=1043.453,262.346,-107.514,171.609,40.293,157.669
C01357=1043.461,262.633,-107.548,171.613,40.296,157.670
C01358=1043.468,262.919,-107.583,171.616,40.298,157.670
C01359=1043.476,263.207,-107.617,171.619,40.301,157.671
C01360=1043.483,263.493,-107.652,171.622,40.303,157.672
C01361=1043.490,263.741,-107.682,171.626,40.306,157.672
C01362=1043.496,263.989,-107.712,171.628,40.308,157.673
C01363=1043.503,264.238,-107.742,171.631,40.310,157.674
C01364=1043.510,264.485,-107.772,171.635,40.313,157.674
C01365=1043.516,264.734,-107.803,171.637,40.315,157.675
C01366=1043.522,264.982,-107.832,171.640,40.317,157.675
C01367=1043.530,265.230,-107.862,171.644,40.319,157.676
C01368=1043.535,265.478,-107.892,171.646,40.321,157.677
C01369=1043.543,265.726,-107.922,171.649,40.324,157.677
C01370=1043.550,265.974,-107.953,171.653,40.326,157.678
C01371=1043.556,266.222,-107.983,171.655,40.329,157.679
C01372=1043.563,266.470,-108.013,171.658,40.331,157.679
C01373=1043.569,266.718,-108.043,171.662,40.333,157.680
C01374=1043.576,266.966,-108.074,171.664,40.335,157.680
C01375=1043.583,267.215,-108.104,171.667,40.337,157.681
C01376=1043.589,267.462,-108.133,171.670,40.339,157.682
C01377=1043.596,267.711,-108.164,171.673,40.342,157.682
C01378=1043.603,267.959,-108.194,171.676,40.344,157.683
C01379=1043.609,268.207,-108.225,171.680,40.347,157.684
C01380=1043.616,268.455,-108.255,171.682,40.349,157.684
C01381=1043.622,268.703,-108.285,171.685,40.351,157.685
C01382=1043.629,268.951,-108.315,171.688,40.353,157.685
C01383=1043.635,269.199,-108.346,171.691,40.355,157.686
C01384=1043.642,269.447,-108.376,171.695,40.358,157.687
C01385=1043.648,269.695,-108.406,171.698,40.360,157.687
C01386=1043.655,269.944,-108.437,171.700,40.362,157.688
C01387=1043.662,270.191,-108.468,171.704,40.365,157.689
C01388=1043.669,270.439,-108.498,171.706,40.367,157.689
C01389=1043.675,270.688,-108.528,171.709,40.369,157.690
C01390=1043.682,270.936,-108.559,171.713,40.372,157.690
C01391=1043.688,271.184,-108.589,171.715,40.374,157.691
C01392=1043.696,271.431,-108.620,171.719,40.376,157.692
C01393=1043.702,271.680,-108.650,171.722,40.378,157.692
C01394=1043.709,271.927,-108.680,171.725,40.381,157.693
C01395=1043.715,272.176,-108.711,171.728,40.383,157.694
C01396=1043.722,272.424,-108.742,171.731,40.385,157.694
C01397=1043.729,272.672,-108.772,171.734,40.387,157.695
C01398=1043.735,272.920,-108.803,171.737,40.390,157.696
C01399=1043.741,273.168,-108.834,171.741,40.392,157.696
C01400=1043.749,273.416,-108.864,171.744,40.395,157.697
C01401=1043.754,273.664,-108.895,171.746,40.397,157.697
C01402=1043.761,273.912,-108.926,171.750,40.400,157.698
C01403=1043.768,274.160,-108.956,171.753,40.402,157.699
C01404=1043.775,274.408,-108.988,171.756,40.404,157.699
C01405=1043.781,274.655,-109.018,171.759,40.406,157.700
C01406=1043.788,274.904,-109.048,171.763,40.409,157.701
C01407=1043.795,275.152,-109.080,171.765,40.411,157.701
C01408=1043.801,275.400,-109.110,171.768,40.413,157.702
C01409=1043.808,275.648,-109.142,171.772,40.416,157.703
C01410=1043.814,275.896,-109.172,171.774,40.418,157.703
C01411=1043.821,276.143,-109.203,171.778,40.420,157.704
C01412=1043.828,276.392,-109.234,171.781,40.423,157.705
C01413=1043.835,276.683,-109.270,171.785,40.426,157.705
C01414=1043.844,276.974,-109.307,171.788,40.428,157.706
C01415=1043.851,277.266,-109.343,171.792,40.431,157.707
C01416=1043.859,277.556,-109.379,171.796,40.434,157.708
C01417=1043.866,277.804,-109.411,171.799,40.436,157.708
C01418=1043.873,278.053,-109.441,171.803,40.439,157.709
C01419=1043.880,278.300,-109.472,171.805,40.441,157.710
C01420=1043.886,278.549,-109.503,171.809,40.443,157.710
C01421=1043.892,278.796,-109.534,171.812,40.446,157.711
C01422=1043.899,279.044,-109.565,171.815,40.448,157.712
C01423=1043.905,279.293,-109.596,171.818,40.450,157.712
C01424=1043.912,279.541,-109.627,171.822,40.453,157.713
C01425=1043.919,279.788,-109.659,171.824,40.455,157.714
C01426=1043.925,280.036,-109.690,171.828,40.458,157.714
C01427=1043.932,280.284,-109.722,171.831,40.460,157.715
C01428=1043.938,280.532,-109.752,171.835,40.463,157.716
C01429=1043.945,280.780,-109.784,171.837,40.465,157.716
C01430=1043.951,281.028,-109.815,171.841,40.467,157.717
C01431=1043.958,281.276,-109.846,171.845,40.470,157.718
C01432=1043.965,281.524,-109.878,171.848,40.472,157.719
C01433=1043.972,281.772,-109.909,171.851,40.474,157.719
C01434=1043.978,282.020,-109.940,171.854,40.477,157.720
C01435=1043.985,282.268,-109.971,171.858,40.479,157.721
C01436=1043.991,282.516,-110.003,171.860,40.482,157.721
C01437=1043.998,282.764,-110.034,171.864,40.484,157.722
C01438=1044.005,283.012,-110.066,171.867,40.486,157.722
C01439=1044.012,283.260,-110.097,171.871,40.489,157.723
C01440=1044.018,283.508,-110.129,171.873,40.491,157.724
C01441=1044.025,283.755,-110.160,171.877,40.494,157.725
C01442=1044.032,284.003,-110.191,171.881,40.496,157.725
C01443=1044.038,284.251,-110.223,171.883,40.499,157.726
C01444=1044.045,284.499,-110.254,171.887,40.501,157.727
C01445=1044.052,284.747,-110.286,171.890,40.504,157.727
C01446=1044.059,284.995,-110.317,171.894,40.506,157.728
C01447=1044.065,285.243,-110.349,171.897,40.508,157.729
C01448=1044.072,285.491,-110.380,171.900,40.511,157.729
C01449=1044.079,285.739,-110.412,171.904,40.513,157.730
C01450=1044.086,285.987,-110.443,171.907,40.516,157.731
C01451=1044.092,286.234,-110.474,171.910,40.518,157.731
C01452=1044.099,286.482,-110.507,171.914,40.520,157.732
C01453=1044.106,286.730,-110.538,171.917,40.523,157.733
C01454=1044.113,286.978,-110.569,171.920,40.525,157.733
C01455=1044.120,287.225,-110.601,171.923,40.528,157.734
C01456=1044.125,287.474,-110.633,171.927,40.531,157.735
C01457=1044.132,287.722,-110.664,171.931,40.533,157.736
C01458=1044.139,287.969,-110.696,171.934,40.536,157.736
C01459=1044.146,288.217,-110.728,171.937,40.538,157.737
C01460=1044.153,288.465,-110.759,171.941,40.540,157.738
C01461=1044.159,288.712,-110.792,171.944,40.543,157.739
C01462=1044.166,288.960,-110.823,171.948,40.545,157.739
C01463=1044.173,289.209,-110.855,171.950,40.548,157.740
C01464=1044.180,289.456,-110.887,171.954,40.551,157.741
C01465=1044.186,289.704,-110.919,171.958,40.553,157.741
C01466=1044.193,289.952,-110.951,171.961,40.555,157.742
C01467=1044.200,290.199,-110.983,171.964,40.558,157.743
C01468=1044.206,290.448,-111.015,171.968,40.560,157.743
C01469=1044.215,290.751,-111.053,171.972,40.564,157.744
C01470=1044.223,291.053,-111.093,171.976,40.567,157.745
C01471=1044.231,291.357,-111.132,171.981,40.569,157.746
C01472=1044.239,291.659,-111.172,171.985,40.573,157.747
C01473=1044.246,291.907,-111.203,171.988,40.575,157.748
C01474=1044.252,292.155,-111.236,171.992,40.578,157.748
C01475=1044.259,292.403,-111.267,171.995,40.580,157.749
C01476=1044.266,292.650,-111.299,171.999,40.583,157.750
C01477=1044.273,292.899,-111.332,172.002,40.586,157.751
C01478=1044.280,293.146,-111.364,172.006,40.588,157.751
C01479=1044.287,293.394,-111.396,172.009,40.590,157.752
C01480=1044.293,293.642,-111.428,172.012,40.593,157.753
C01481=1044.300,293.889,-111.460,172.016,40.596,157.754
C01482=1044.306,294.138,-111.493,172.020,40.598,157.754
C01483=1044.313,294.385,-111.525,172.023,40.601,157.755
C01484=1044.320,294.633,-111.558,172.026,40.603,157.756
C01485=1044.326,294.881,-111.589,172.030,40.606,157.756
C01486=1044.333,295.128,-111.622,172.034,40.609,157.757
C01487=1044.340,295.376,-111.654,172.037,40.611,157.758
C01488=1044.347,295.624,-111.687,172.040,40.613,157.759
C01489=1044.353,295.872,-111.718,172.044,40.616,157.759
C01490=1044.360,296.119,-111.751,172.048,40.619,157.760
C01491=1044.367,296.368,-111.784,172.051,40.622,157.761
C01492=1044.373,296.615,-111.817,172.055,40.624,157.762
C01493=1044.380,296.863,-111.849,172.059,40.627,157.762
C01494=1044.386,297.110,-111.882,172.062,40.630,157.763
C01495=1044.392,297.358,-111.915,172.065,40.632,157.764
C01496=1044.399,297.606,-111.948,172.069,40.635,157.765
C01497=1044.406,297.853,-111.980,172.073,40.638,157.766
C01498=1044.413,298.101,-112.013,172.076,40.640,157.766
C01499=1044.420,298.349,-112.046,172.080,40.643,157.767
C01500=1044.426,298.597,-112.079,172.083,40.646,157.768
C01501=1044.432,298.844,-112.111,172.087,40.648,157.769
C01502=1044.439,299.092,-112.143,172.091,40.651,157.769
C01503=1044.446,299.340,-112.177,172.094,40.654,157.770
C01504=1044.452,299.588,-112.209,172.098,40.656,157.771
C01505=1044.459,299.835,-112.242,172.101,40.659,157.772
C01506=1044.466,300.083,-112.275,172.105,40.662,157.772
C01507=1044.473,300.331,-112.307,172.108,40.665,157.773
C01508=1044.479,300.578,-112.340,172.112,40.667,157.774
C01509=1044.486,300.827,-112.373,172.116,40.670,157.775
C01510=1044.492,301.074,-112.406,172.120,40.673,157.776
C01511=1044.498,301.322,-112.439,172.123,40.675,157.776
C01512=1044.506,301.569,-112.472,172.126,40.679,157.777
C01513=1044.513,301.817,-112.505,172.130,40.681,157.778
C01514=1044.519,302.065,-112.538,172.134,40.684,157.779
C01515=1044.526,302.313,-112.570,172.138,40.687,157.780
C01516=1044.532,302.560,-112.603,172.142,40.689,157.780
C01517=1044.539,302.808,-112.637,172.146,40.692,157.781
C01518=1044.546,303.055,-112.669,172.148,40.695,157.782
C01519=1044.553,303.304,-112.702,172.152,40.697,157.783
C01520=1044.560,303.550,-112.736,172.156,40.700,157.783
C01521=1044.567,303.799,-112.769,172.160,40.703,157.784
C01522=1044.573,304.046,-112.802,172.164,40.705,157.785
C01523=1044.580,304.293,-112.835,172.168,40.708,157.786
C01524=1044.587,304.541,-112.868,172.172,40.711,157.787
C01525=1044.596,304.861,-112.910,172.176,40.714,157.788
C01526=1044.604,305.180,-112.953,172.181,40.718,157.789
C01527=1044.613,305.499,-112.996,172.186,40.722,157.790
C01528=1044.623,305.818,-113.039,172.191,40.725,157.791
C01529=1044.629,306.066,-113.072,172.194,40.728,157.791
C01530=1044.636,306.314,-113.105,172.198,40.731,157.792
C01531=1044.642,306.561,-113.138,172.202,40.733,157.793
C01532=1044.649,306.810,-113.171,172.206,40.736,157.794
C01533=1044.656,307.057,-113.205,172.209,40.739,157.795
C01534=1044.663,307.305,-113.237,172.213,40.741,157.795
C01535=1044.671,307.552,-113.271,172.217,40.744,157.796
C01536=1044.677,307.799,-113.304,172.221,40.747,157.797
C01537=1044.684,308.048,-113.338,172.225,40.750,157.798
C01538=1044.691,308.295,-113.371,172.229,40.753,157.799
C01539=1044.698,308.543,-113.404,172.233,40.755,157.800
C01540=1044.705,308.790,-113.438,172.237,40.758,157.800
C01541=1044.711,309.037,-113.471,172.240,40.761,157.801
C01542=1044.719,309.285,-113.504,172.244,40.764,157.802
C01543=1044.726,309.533,-113.538,172.248,40.766,157.803
C01544=1044.733,309.781,-113.571,172.252,40.770,157.804
C01545=1044.740,310.028,-113.604,172.256,40.772,157.804
C01546=1044.747,310.276,-113.638,172.260,40.775,157.805
C01547=1044.754,310.523,-113.672,172.264,40.777,157.806
C01548=1044.760,310.771,-113.705,172.268,40.781,157.807
C01549=1044.768,311.019,-113.739,172.272,40.783,157.808
C01550=1044.775,311.267,-113.772,172.275,40.786,157.809
C01551=1044.781,311.514,-113.806,172.279,40.789,157.809
C01552=1044.789,311.762,-113.838,172.283,40.792,157.810
C01553=1044.796,312.009,-113.872,172.287,40.794,157.811
C01554=1044.804,312.257,-113.906,172.291,40.797,157.812
C01555=1044.811,312.505,-113.940,172.295,40.800,157.813
C01556=1044.817,312.752,-113.974,172.299,40.803,157.814
C01557=1044.824,313.000,-114.008,172.303,40.806,157.814
C01558=1044.830,313.248,-114.042,172.307,40.809,157.815
C01559=1044.837,313.495,-114.076,172.311,40.812,157.816
C01560=1044.844,313.742,-114.109,172.315,40.815,157.817
C01561=1044.850,313.990,-114.144,172.319,40.818,157.818
C01562=1044.857,314.237,-114.177,172.323,40.821,157.819
C01563=1044.864,314.485,-114.212,172.327,40.824,157.820
C01564=1044.871,314.733,-114.246,172.331,40.827,157.821
C01565=1044.878,314.980,-114.281,172.335,40.830,157.821
C01566=1044.884,315.227,-114.314,172.338,40.833,157.822
C01567=1044.891,315.475,-114.349,172.342,40.836,157.823
C01568=1044.898,315.723,-114.382,172.346,40.839,157.824
C01569=1044.904,315.971,-114.417,172.350,40.842,157.825
C01570=1044.911,316.218,-114.450,172.354,40.845,157.826
C01571=1044.918,316.465,-114.485,172.358,40.848,157.827
C01572=1044.925,316.713,-114.519,172.362,40.851,157.828
C01573=1044.931,316.961,-114.554,172.366,40.854,157.828
C01574=1044.939,317.208,-114.588,172.370,40.857,157.829
C01575=1044.945,317.455,-114.622,172.374,40.860,157.830
C01576=1044.952,317.703,-114.656,172.378,40.863,157.831
C01577=1044.958,317.951,-114.690,172.382,40.866,157.832
C01578=1044.966,318.198,-114.725,172.386,40.869,157.833
C01579=1044.972,318.446,-114.759,172.390,40.872,157.834
C01580=1044.980,318.693,-114.794,172.394,40.875,157.835
C01581=1044.988,319.017,-114.839,172.399,40.880,157.836
C01582=1044.998,319.341,-114.884,172.405,40.883,157.837
C01583=1045.007,319.664,-114.929,172.410,40.888,157.838
C01584=1045.016,319.989,-114.974,172.416,40.891,157.839
C01585=1045.023,320.236,-115.008,172.420,40.894,157.840
C01586=1045.030,320.484,-115.043,172.424,40.897,157.841
C01587=1045.037,320.731,-115.077,172.428,40.901,157.842
C01588=1045.044,320.979,-115.112,172.432,40.903,157.843
C01589=1045.050,321.227,-115.147,172.436,40.907,157.844
C01590=1045.058,321.474,-115.181,172.440,40.910,157.845
C01591=1045.064,321.722,-115.216,172.445,40.913,157.846
C01592=1045.072,321.969,-115.250,172.449,40.916,157.847
C01593=1045.078,322.216,-115.285,172.453,40.919,157.848
C01594=1045.085,322.464,-115.319,172.457,40.922,157.849
C01595=1045.092,322.711,-115.354,172.461,40.925,157.849
C01596=1045.099,322.959,-115.388,172.465,40.928,157.850
C01597=1045.106,323.206,-115.423,172.470,40.931,157.851
C01598=1045.113,323.454,-115.458,172.474,40.934,157.852
C01599=1045.121,323.701,-115.493,172.478,40.938,157.853
C01600=1045.127,323.949,-115.527,172.482,40.941,157.854
C01601=1045.134,324.196,-115.562,172.486,40.944,157.855
C01602=1045.141,324.443,-115.597,172.492,40.947,157.856
C01603=1045.149,324.691,-115.632,172.496,40.950,157.857
C01604=1045.156,324.939,-115.666,172.500,40.953,157.858
C01605=1045.163,325.186,-115.702,172.504,40.957,157.859
C01606=1045.170,325.433,-115.736,172.508,40.960,157.860
C01607=1045.177,325.681,-115.771,172.513,40.963,157.861
C01608=1045.184,325.928,-115.806,172.517,40.966,157.862
C01609=1045.192,326.176,-115.841,172.521,40.969,157.863
C01610=1045.198,326.424,-115.876,172.525,40.972,157.863
C01611=1045.206,326.671,-115.910,172.530,40.976,157.864
C01612=1045.212,326.918,-115.945,172.534,40.979,157.865
C01613=1045.221,327.166,-115.980,172.538,40.982,157.866
C01614=1045.227,327.413,-116.015,172.542,40.985,157.867
C01615=1045.234,327.661,-116.051,172.547,40.988,157.868
C01616=1045.242,327.908,-116.085,172.551,40.991,157.869
C01617=1045.249,328.156,-116.121,172.555,40.995,157.870
C01618=1045.256,328.403,-116.156,172.560,40.998,157.871
C01619=1045.263,328.650,-116.190,172.564,41.001,157.872
C01620=1045.271,328.898,-116.226,172.568,41.004,157.873
C01621=1045.278,329.145,-116.260,172.573,41.008,157.874
C01622=1045.285,329.392,-116.296,172.578,41.011,157.875
C01623=1045.293,329.640,-116.332,172.582,41.014,157.876
C01624=1045.299,329.888,-116.367,172.586,41.017,157.877
C01625=1045.306,330.135,-116.402,172.591,41.021,157.878
C01626=1045.313,330.382,-116.438,172.595,41.024,157.879
C01627=1045.321,330.630,-116.473,172.599,41.027,157.880
C01628=1045.327,330.877,-116.508,172.604,41.031,157.881
C01629=1045.334,331.124,-116.544,172.608,41.034,157.882
C01630=1045.342,331.372,-116.580,172.612,41.037,157.883
C01631=1045.349,331.619,-116.615,172.617,41.041,157.884
C01632=1045.356,331.866,-116.651,172.622,41.044,157.885
C01633=1045.363,332.114,-116.686,172.626,41.048,157.886
C01634=1045.370,332.361,-116.721,172.630,41.051,157.887
C01635=1045.377,332.608,-116.757,172.635,41.054,157.888
C01636=1045.384,332.856,-116.793,172.639,41.058,157.889
C01637=1045.393,333.175,-116.839,172.645,41.062,157.890
C01638=1045.402,333.495,-116.885,172.651,41.067,157.892
C01639=1045.412,333.813,-116.931,172.657,41.071,157.893
C01640=1045.421,334.132,-116.978,172.663,41.075,157.894
C01641=1045.428,334.380,-117.013,172.667,41.079,157.895
C01642=1045.435,334.626,-117.049,172.671,41.082,157.896
C01643=1045.442,334.874,-117.085,172.676,41.085,157.897
C01644=1045.449,335.121,-117.120,172.681,41.089,157.898
C01645=1045.457,335.369,-117.156,172.685,41.092,157.899
C01646=1045.463,335.616,-117.192,172.690,41.096,157.901
C01647=1045.471,335.863,-117.228,172.694,41.099,157.901
C01648=1045.478,336.110,-117.264,172.699,41.103,157.903
C01649=1045.485,336.358,-117.300,172.704,41.106,157.904
C01650=1045.492,336.605,-117.336,172.709,41.109,157.905
C01651=1045.500,336.853,-117.372,172.713,41.113,157.906
C01652=1045.506,337.100,-117.408,172.717,41.117,157.907
C01653=1045.514,337.347,-117.444,172.722,41.120,157.908
C01654=1045.521,337.594,-117.480,172.726,41.124,157.909
C01655=1045.528,337.841,-117.517,172.732,41.127,157.910
C01656=1045.535,338.089,-117.553,172.736,41.131,157.911
C01657=1045.542,338.336,-117.589,172.741,41.135,157.912
C01658=1045.550,338.583,-117.625,172.745,41.138,157.913
C01659=1045.556,338.831,-117.661,172.749,41.142,157.914
C01660=1045.564,339.079,-117.697,172.755,41.145,157.915
C01661=1045.571,339.326,-117.734,172.759,41.149,157.916
C01662=1045.578,339.573,-117.770,172.764,41.153,157.918
C01663=1045.586,339.820,-117.807,172.768,41.156,157.919
C01664=1045.593,340.067,-117.843,172.773,41.159,157.920
C01665=1045.600,340.314,-117.880,172.778,41.163,157.921
C01666=1045.607,340.562,-117.916,172.783,41.167,157.922
C01667=1045.615,340.809,-117.952,172.787,41.170,157.923
C01668=1045.621,341.056,-117.988,172.792,41.174,157.924
C01669=1045.629,341.304,-118.025,172.797,41.178,157.925
C01670=1045.637,341.551,-118.061,172.802,41.181,157.926
C01671=1045.643,341.798,-118.098,172.806,41.185,157.927
C01672=1045.651,342.045,-118.134,172.811,41.189,157.929
C01673=1045.659,342.293,-118.171,172.817,41.192,157.930
C01674=1045.665,342.540,-118.207,172.821,41.196,157.931
C01675=1045.673,342.786,-118.244,172.826,41.200,157.932
C01676=1045.680,343.034,-118.281,172.831,41.203,157.933
C01677=1045.687,343.282,-118.318,172.836,41.207,157.934
C01678=1045.694,343.528,-118.354,172.840,41.211,157.935
C01679=1045.701,343.776,-118.391,172.845,41.215,157.936
C01680=1045.709,344.023,-118.428,172.850,41.218,157.938
C01681=1045.716,344.270,-118.465,172.855,41.222,157.939
C01682=1045.724,344.517,-118.502,172.860,41.226,157.940
C01683=1045.731,344.764,-118.538,172.864,41.229,157.941
C01684=1045.738,345.011,-118.576,172.870,41.234,157.942
C01685=1045.745,345.259,-118.612,172.874,41.237,157.943
C01686=1045.753,345.506,-118.649,172.879,41.241,157.944
C01687=1045.760,345.753,-118.685,172.885,41.244,157.946
C01688=1045.767,346.000,-118.723,172.889,41.249,157.947
C01689=1045.774,346.248,-118.759,172.894,41.252,157.948
C01690=1045.782,346.494,-118.796,172.899,41.256,157.949
C01691=1045.789,346.742,-118.834,172.904,41.260,157.950
C01692=1045.796,346.989,-118.871,172.909,41.264,157.951
C01693=1045.805,347.275,-118.913,172.915,41.268,157.953
C01694=1045.813,347.561,-118.957,172.920,41.273,157.954
C01695=1045.822,347.847,-118.999,172.926,41.277,157.956
C01696=1045.830,348.132,-119.042,172.933,41.281,157.957
C01697=1045.837,348.380,-119.080,172.937,41.286,157.958
C01698=1045.845,348.626,-119.117,172.942,41.289,157.959
C01699=1045.853,348.874,-119.154,172.948,41.293,157.961
C01700=1045.860,349.121,-119.191,172.952,41.297,157.962
C01701=1045.868,349.368,-119.228,172.957,41.301,157.963
C01702=1045.875,349.615,-119.266,172.963,41.305,157.964
C01703=1045.882,349.862,-119.303,172.967,41.309,157.965
C01704=1045.890,350.109,-119.340,172.972,41.313,157.966
C01705=1045.897,350.356,-119.378,172.978,41.317,157.968
C01706=1045.904,350.604,-119.415,172.982,41.321,157.969
C01707=1045.912,350.851,-119.453,172.988,41.325,157.970
C01708=1045.919,351.098,-119.490,172.993,41.329,157.971
C01709=1045.927,351.346,-119.528,172.998,41.332,157.973
C01710=1045.934,351.593,-119.566,173.003,41.337,157.974
C01711=1045.942,351.839,-119.604,173.008,41.341,157.975
C01712=1045.949,352.086,-119.642,173.014,41.345,157.976
C01713=1045.956,352.334,-119.679,173.019,41.349,157.977
C01714=1045.963,352.581,-119.717,173.023,41.353,157.979
C01715=1045.971,352.828,-119.753,173.029,41.357,157.980
C01716=1045.979,353.074,-119.792,173.034,41.361,157.981
C01717=1045.986,353.321,-119.829,173.040,41.365,157.983
C01718=1045.993,353.568,-119.867,173.044,41.369,157.984
C01719=1046.001,353.815,-119.905,173.050,41.373,157.985
C01720=1046.009,354.063,-119.943,173.055,41.377,157.986
C01721=1046.016,354.310,-119.980,173.061,41.381,157.988
C01722=1046.024,354.556,-120.019,173.066,41.385,157.989
C01723=1046.031,354.803,-120.056,173.070,41.390,157.990
C01724=1046.038,355.050,-120.094,173.076,41.394,157.991
C01725=1046.046,355.298,-120.132,173.081,41.398,157.993
C01726=1046.054,355.544,-120.171,173.087,41.402,157.994
C01727=1046.061,355.791,-120.208,173.092,41.406,157.995
C01728=1046.069,356.038,-120.246,173.098,41.410,157.997
C01729=1046.076,356.286,-120.284,173.102,41.415,157.998
C01730=1046.084,356.532,-120.323,173.108,41.419,157.999
C01731=1046.091,356.779,-120.360,173.113,41.423,158.000
C01732=1046.099,357.027,-120.399,173.119,41.427,158.002
C01733=1046.107,357.273,-120.437,173.124,41.431,158.003
C01734=1046.114,357.520,-120.474,173.130,41.436,158.004
C01735=1046.121,357.767,-120.513,173.135,41.440,158.006
C01736=1046.129,358.014,-120.552,173.140,41.444,158.007
C01737=1046.136,358.261,-120.589,173.145,41.448,158.008
C01738=1046.144,358.508,-120.628,173.151,41.453,158.010
C01739=1046.152,358.755,-120.666,173.156,41.457,158.011
C01740=1046.160,359.002,-120.704,173.162,41.461,158.012
C01741=1046.166,359.249,-120.743,173.168,41.466,158.014
C01742=1046.175,359.496,-120.782,173.173,41.470,158.015
C01743=1046.182,359.742,-120.820,173.179,41.474,158.016
C01744=1046.190,359.990,-120.858,173.184,41.479,158.018
C01745=1046.197,360.237,-120.896,173.190,41.483,158.019
C01746=1046.204,360.483,-120.935,173.195,41.487,158.020
C01747=1046.212,360.731,-120.974,173.201,41.492,158.022
C01748=1046.222,361.035,-121.022,173.208,41.497,158.023
C01749=1046.234,361.415,-121.081,173.216,41.503,158.026
C01750=1046.244,361.736,-121.132,173.223,41.509,158.027
C01751=1046.254,362.056,-121.181,173.230,41.515,158.029
C01752=1046.264,362.377,-121.231,173.237,41.521,158.031
C01753=1046.271,362.625,-121.270,173.243,41.525,158.032
C01754=1046.279,362.870,-121.309,173.249,41.530,158.034
C01755=1046.287,363.118,-121.348,173.254,41.535,158.035
C01756=1046.294,363.364,-121.387,173.260,41.539,158.036
C01757=1046.303,363.611,-121.426,173.266,41.543,158.038
C01758=1046.309,363.858,-121.465,173.271,41.548,158.039
C01759=1046.317,364.105,-121.504,173.277,41.553,158.041
C01760=1046.325,364.351,-121.543,173.282,41.557,158.042
C01761=1046.333,364.599,-121.582,173.288,41.561,158.044
C01762=1046.340,364.845,-121.621,173.294,41.566,158.045
C01763=1046.347,365.092,-121.661,173.299,41.571,158.046
C01764=1046.356,365.339,-121.700,173.306,41.575,158.048
C01765=1046.363,365.586,-121.739,173.312,41.580,158.049
C01766=1046.371,365.832,-121.778,173.318,41.585,158.051
C01767=1046.378,366.080,-121.817,173.323,41.589,158.052
C01768=1046.386,366.326,-121.856,173.329,41.594,158.054
C01769=1046.394,366.573,-121.895,173.335,41.598,158.055
C01770=1046.402,366.820,-121.935,173.340,41.603,158.057
C01771=1046.409,367.066,-121.974,173.346,41.608,158.058
C01772=1046.417,367.313,-122.013,173.352,41.612,158.060
C01773=1046.425,367.560,-122.053,173.357,41.617,158.061
C01774=1046.433,367.806,-122.092,173.364,41.622,158.063
C01775=1046.441,368.053,-122.132,173.370,41.626,158.064
C01776=1046.448,368.300,-122.172,173.376,41.631,158.065
C01777=1046.457,368.547,-122.210,173.381,41.635,158.067
C01778=1046.464,368.794,-122.250,173.387,41.640,158.068
C01779=1046.472,369.040,-122.289,173.393,41.645,158.070
C01780=1046.480,369.287,-122.329,173.400,41.650,158.071
C01781=1046.488,369.533,-122.368,173.405,41.654,158.073
C01782=1046.496,369.780,-122.408,173.411,41.659,158.074
C01783=1046.505,370.027,-122.448,173.417,41.664,158.076
C01784=1046.512,370.274,-122.488,173.423,41.669,158.077
C01785=1046.519,370.520,-122.527,173.429,41.673,158.079
C01786=1046.528,370.767,-122.566,173.435,41.679,158.081
C01787=1046.536,371.013,-122.606,173.441,41.683,158.082
C01788=1046.543,371.260,-122.646,173.447,41.688,158.084
C01789=1046.552,371.507,-122.686,173.454,41.693,158.085
C01790=1046.559,371.754,-122.725,173.459,41.698,158.087
C01791=1046.567,372.000,-122.766,173.465,41.703,158.088
C01792=1046.575,372.247,-122.806,173.471,41.708,158.090
C01793=1046.583,372.494,-122.846,173.478,41.712,158.091
C01794=1046.591,372.741,-122.886,173.484,41.718,158.093
C01795=1046.598,372.986,-122.926,173.490,41.723,158.095
C01796=1046.606,373.233,-122.966,173.495,41.727,158.096
C01797=1046.614,373.480,-123.007,173.502,41.732,158.098
C01798=1046.622,373.726,-123.046,173.508,41.738,158.099
C01799=1046.630,373.973,-123.086,173.514,41.743,158.101
C01800=1046.638,374.219,-123.127,173.521,41.747,158.102
C01801=1046.646,374.466,-123.166,173.527,41.752,158.104
C01802=1046.654,374.713,-123.207,173.533,41.758,158.106
C01803=1046.661,374.960,-123.247,173.540,41.763,158.107
C01804=1046.670,375.207,-123.288,173.545,41.768,158.109
C01805=1046.681,375.546,-123.344,173.554,41.774,158.111
